    ! Character: O
    PROC char_upperO()
        VAR robtarget pTarget;
        pTarget:=refTarget;
        pTarget.trans:=[12,32.0,0];
        MoveL pTarget,vSpeed,fine,tTool\WObj:=wWobj;
        Set do_pen;
        pTarget.trans:=[9,31.0,0];
        MoveL pTarget,vSpeed,z0,tTool\WObj:=wWobj;
        pTarget.trans:=[7,29.0,0];
        MoveL pTarget,vSpeed,z0,tTool\WObj:=wWobj;
        pTarget.trans:=[5,26.0,0];
        MoveL pTarget,vSpeed,z0,tTool\WObj:=wWobj;
        pTarget.trans:=[4,24.0,0];
        MoveL pTarget,vSpeed,z0,tTool\WObj:=wWobj;
        pTarget.trans:=[3,20.0,0];
        MoveL pTarget,vSpeed,z0,tTool\WObj:=wWobj;
        pTarget.trans:=[3,16.0,0];
        MoveL pTarget,vSpeed,z0,tTool\WObj:=wWobj;
        pTarget.trans:=[4,13.0,0];
        MoveL pTarget,vSpeed,z0,tTool\WObj:=wWobj;
        pTarget.trans:=[5,12.0,0];
        MoveL pTarget,vSpeed,z0,tTool\WObj:=wWobj;
        pTarget.trans:=[7,11.0,0];
        MoveL pTarget,vSpeed,z0,tTool\WObj:=wWobj;
        pTarget.trans:=[9,11.0,0];
        MoveL pTarget,vSpeed,z0,tTool\WObj:=wWobj;
        pTarget.trans:=[12,12.0,0];
        MoveL pTarget,vSpeed,z0,tTool\WObj:=wWobj;
        pTarget.trans:=[14,14.0,0];
        MoveL pTarget,vSpeed,z0,tTool\WObj:=wWobj;
        pTarget.trans:=[16,17.0,0];
        MoveL pTarget,vSpeed,z0,tTool\WObj:=wWobj;
        pTarget.trans:=[17,19.0,0];
        MoveL pTarget,vSpeed,z0,tTool\WObj:=wWobj;
        pTarget.trans:=[18,23.0,0];
        MoveL pTarget,vSpeed,z0,tTool\WObj:=wWobj;
        pTarget.trans:=[18,27.0,0];
        MoveL pTarget,vSpeed,z0,tTool\WObj:=wWobj;
        pTarget.trans:=[17,30.0,0];
        MoveL pTarget,vSpeed,z0,tTool\WObj:=wWobj;
        pTarget.trans:=[16,31.0,0];
        MoveL pTarget,vSpeed,z0,tTool\WObj:=wWobj;
        pTarget.trans:=[14,32.0,0];
        MoveL pTarget,vSpeed,z0,tTool\WObj:=wWobj;
        pTarget.trans:=[12,32.0,0];
        MoveL pTarget,vSpeed,z0,tTool\WObj:=wWobj;
        pTarget.trans:=[10,30.0,0];
        MoveL pTarget,vSpeed,z0,tTool\WObj:=wWobj;
        pTarget.trans:=[10,27.0,0];
        MoveL pTarget,vSpeed,z0,tTool\WObj:=wWobj;
        pTarget.trans:=[11,24.0,0];
        MoveL pTarget,vSpeed,z0,tTool\WObj:=wWobj;
        pTarget.trans:=[13,21.0,0];
        MoveL pTarget,vSpeed,z0,tTool\WObj:=wWobj;
        pTarget.trans:=[15,19.0,0];
        MoveL pTarget,vSpeed,z0,tTool\WObj:=wWobj;
        pTarget.trans:=[18,17.0,0];
        MoveL pTarget,vSpeed,z0,tTool\WObj:=wWobj;
        pTarget.trans:=[20,16.0,0];
        MoveL pTarget,vSpeed,fine,tTool\WObj:=wWobj;
        Reset do_pen;
        MoveL RelTool(pTarget,0,0,-2),vSpeed,z0,tTool\WObj:=wWobj;
        wWobj.oframe.trans.x:=wWobj.oframe.trans.x+17;
    ENDPROC

    ! Character: P
    PROC char_upperP()
        VAR robtarget pTarget;
        pTarget:=refTarget;
        pTarget.trans:=[13,30.0,0];
        MoveL pTarget,vSpeed,fine,tTool\WObj:=wWobj;
        Set do_pen;
        pTarget.trans:=[14,29.0,0];
        MoveL pTarget,vSpeed,z0,tTool\WObj:=wWobj;
        pTarget.trans:=[14,26.0,0];
        MoveL pTarget,vSpeed,z0,tTool\WObj:=wWobj;
        pTarget.trans:=[13,22.0,0];
        MoveL pTarget,vSpeed,z0,tTool\WObj:=wWobj;
        pTarget.trans:=[12,19.0,0];
        MoveL pTarget,vSpeed,z0,tTool\WObj:=wWobj;
        pTarget.trans:=[11,17.0,0];
        MoveL pTarget,vSpeed,z0,tTool\WObj:=wWobj;
        pTarget.trans:=[9,14.0,0];
        MoveL pTarget,vSpeed,z0,tTool\WObj:=wWobj;
        pTarget.trans:=[7,12.0,0];
        MoveL pTarget,vSpeed,z0,tTool\WObj:=wWobj;
        pTarget.trans:=[5,11.0,0];
        MoveL pTarget,vSpeed,z0,tTool\WObj:=wWobj;
        pTarget.trans:=[4,11.0,0];
        MoveL pTarget,vSpeed,z0,tTool\WObj:=wWobj;
        pTarget.trans:=[3,12.0,0];
        MoveL pTarget,vSpeed,z0,tTool\WObj:=wWobj;
        pTarget.trans:=[3,15.0,0];
        MoveL pTarget,vSpeed,z0,tTool\WObj:=wWobj;
        pTarget.trans:=[4,20.0,0];
        MoveL pTarget,vSpeed,z0,tTool\WObj:=wWobj;
        pTarget.trans:=[5,23.0,0];
        MoveL pTarget,vSpeed,z0,tTool\WObj:=wWobj;
        pTarget.trans:=[6,25.0,0];
        MoveL pTarget,vSpeed,z0,tTool\WObj:=wWobj;
        pTarget.trans:=[8,28.0,0];
        MoveL pTarget,vSpeed,z0,tTool\WObj:=wWobj;
        pTarget.trans:=[10,30.0,0];
        MoveL pTarget,vSpeed,z0,tTool\WObj:=wWobj;
        pTarget.trans:=[12,31.0,0];
        MoveL pTarget,vSpeed,z0,tTool\WObj:=wWobj;
        pTarget.trans:=[15,32.0,0];
        MoveL pTarget,vSpeed,z0,tTool\WObj:=wWobj;
        pTarget.trans:=[20,32.0,0];
        MoveL pTarget,vSpeed,z0,tTool\WObj:=wWobj;
        pTarget.trans:=[22,31.0,0];
        MoveL pTarget,vSpeed,z0,tTool\WObj:=wWobj;
        pTarget.trans:=[23,30.0,0];
        MoveL pTarget,vSpeed,z0,tTool\WObj:=wWobj;
        pTarget.trans:=[24,28.0,0];
        MoveL pTarget,vSpeed,z0,tTool\WObj:=wWobj;
        pTarget.trans:=[24,25.0,0];
        MoveL pTarget,vSpeed,z0,tTool\WObj:=wWobj;
        pTarget.trans:=[23,23.0,0];
        MoveL pTarget,vSpeed,z0,tTool\WObj:=wWobj;
        pTarget.trans:=[22,22.0,0];
        MoveL pTarget,vSpeed,z0,tTool\WObj:=wWobj;
        pTarget.trans:=[20,21.0,0];
        MoveL pTarget,vSpeed,z0,tTool\WObj:=wWobj;
        pTarget.trans:=[17,21.0,0];
        MoveL pTarget,vSpeed,z0,tTool\WObj:=wWobj;
        pTarget.trans:=[15,22.0,0];
        MoveL pTarget,vSpeed,z0,tTool\WObj:=wWobj;
        pTarget.trans:=[14,23.0,0];
        MoveL pTarget,vSpeed,fine,tTool\WObj:=wWobj;
        Reset do_pen;
        MoveL RelTool(pTarget,0,0,-2),vSpeed,z0,tTool\WObj:=wWobj;
        wWobj.oframe.trans.x:=wWobj.oframe.trans.x+21;
    ENDPROC

    ! Character: Q
    PROC char_upperQ()
        VAR robtarget pTarget;
        pTarget:=refTarget;
        pTarget.trans:=[13,26.0,0];
        MoveL pTarget,vSpeed,fine,tTool\WObj:=wWobj;
        Set do_pen;
        pTarget.trans:=[12,24.0,0];
        MoveL pTarget,vSpeed,z0,tTool\WObj:=wWobj;
        pTarget.trans:=[11,23.0,0];
        MoveL pTarget,vSpeed,z0,tTool\WObj:=wWobj;
        pTarget.trans:=[9,22.0,0];
        MoveL pTarget,vSpeed,z0,tTool\WObj:=wWobj;
        pTarget.trans:=[7,22.0,0];
        MoveL pTarget,vSpeed,z0,tTool\WObj:=wWobj;
        pTarget.trans:=[6,24.0,0];
        MoveL pTarget,vSpeed,z0,tTool\WObj:=wWobj;
        pTarget.trans:=[6,26.0,0];
        MoveL pTarget,vSpeed,z0,tTool\WObj:=wWobj;
        pTarget.trans:=[7,29.0,0];
        MoveL pTarget,vSpeed,z0,tTool\WObj:=wWobj;
        pTarget.trans:=[9,31.0,0];
        MoveL pTarget,vSpeed,z0,tTool\WObj:=wWobj;
        pTarget.trans:=[12,32.0,0];
        MoveL pTarget,vSpeed,z0,tTool\WObj:=wWobj;
        pTarget.trans:=[15,32.0,0];
        MoveL pTarget,vSpeed,z0,tTool\WObj:=wWobj;
        pTarget.trans:=[17,31.0,0];
        MoveL pTarget,vSpeed,z0,tTool\WObj:=wWobj;
        pTarget.trans:=[18,29.0,0];
        MoveL pTarget,vSpeed,z0,tTool\WObj:=wWobj;
        pTarget.trans:=[18,25.0,0];
        MoveL pTarget,vSpeed,z0,tTool\WObj:=wWobj;
        pTarget.trans:=[17,22.0,0];
        MoveL pTarget,vSpeed,z0,tTool\WObj:=wWobj;
        pTarget.trans:=[15,19.0,0];
        MoveL pTarget,vSpeed,z0,tTool\WObj:=wWobj;
        pTarget.trans:=[11,15.0,0];
        MoveL pTarget,vSpeed,z0,tTool\WObj:=wWobj;
        pTarget.trans:=[8,13.0,0];
        MoveL pTarget,vSpeed,z0,tTool\WObj:=wWobj;
        pTarget.trans:=[6,12.0,0];
        MoveL pTarget,vSpeed,z0,tTool\WObj:=wWobj;
        pTarget.trans:=[3,11.0,0];
        MoveL pTarget,vSpeed,z0,tTool\WObj:=wWobj;
        pTarget.trans:=[1,11.0,0];
        MoveL pTarget,vSpeed,z0,tTool\WObj:=wWobj;
        pTarget.trans:=[0,12.0,0];
        MoveL pTarget,vSpeed,z0,tTool\WObj:=wWobj;
        pTarget.trans:=[0,14.0,0];
        MoveL pTarget,vSpeed,z0,tTool\WObj:=wWobj;
        pTarget.trans:=[1,15.0,0];
        MoveL pTarget,vSpeed,z0,tTool\WObj:=wWobj;
        pTarget.trans:=[3,15.0,0];
        MoveL pTarget,vSpeed,z0,tTool\WObj:=wWobj;
        pTarget.trans:=[5,14.0,0];
        MoveL pTarget,vSpeed,z0,tTool\WObj:=wWobj;
        pTarget.trans:=[8,12.0,0];
        MoveL pTarget,vSpeed,z0,tTool\WObj:=wWobj;
        pTarget.trans:=[11,11.0,0];
        MoveL pTarget,vSpeed,z0,tTool\WObj:=wWobj;
        pTarget.trans:=[14,11.0,0];
        MoveL pTarget,vSpeed,z0,tTool\WObj:=wWobj;
        pTarget.trans:=[17,12.0,0];
        MoveL pTarget,vSpeed,z0,tTool\WObj:=wWobj;
        pTarget.trans:=[19,14.0,0];
        MoveL pTarget,vSpeed,fine,tTool\WObj:=wWobj;
        Reset do_pen;
        MoveL RelTool(pTarget,0,0,-2),vSpeed,z0,tTool\WObj:=wWobj;
        wWobj.oframe.trans.x:=wWobj.oframe.trans.x+19;
    ENDPROC

    ! Character: R
    PROC char_upperR()
        VAR robtarget pTarget;
        pTarget:=refTarget;
        pTarget.trans:=[13,30.0,0];
        MoveL pTarget,vSpeed,fine,tTool\WObj:=wWobj;
        Set do_pen;
        pTarget.trans:=[14,29.0,0];
        MoveL pTarget,vSpeed,z0,tTool\WObj:=wWobj;
        pTarget.trans:=[14,26.0,0];
        MoveL pTarget,vSpeed,z0,tTool\WObj:=wWobj;
        pTarget.trans:=[13,22.0,0];
        MoveL pTarget,vSpeed,z0,tTool\WObj:=wWobj;
        pTarget.trans:=[12,19.0,0];
        MoveL pTarget,vSpeed,z0,tTool\WObj:=wWobj;
        pTarget.trans:=[11,17.0,0];
        MoveL pTarget,vSpeed,z0,tTool\WObj:=wWobj;
        pTarget.trans:=[9,14.0,0];
        MoveL pTarget,vSpeed,z0,tTool\WObj:=wWobj;
        pTarget.trans:=[7,12.0,0];
        MoveL pTarget,vSpeed,z0,tTool\WObj:=wWobj;
        pTarget.trans:=[5,11.0,0];
        MoveL pTarget,vSpeed,z0,tTool\WObj:=wWobj;
        pTarget.trans:=[4,11.0,0];
        MoveL pTarget,vSpeed,z0,tTool\WObj:=wWobj;
        pTarget.trans:=[3,12.0,0];
        MoveL pTarget,vSpeed,z0,tTool\WObj:=wWobj;
        pTarget.trans:=[3,15.0,0];
        MoveL pTarget,vSpeed,z0,tTool\WObj:=wWobj;
        pTarget.trans:=[4,20.0,0];
        MoveL pTarget,vSpeed,z0,tTool\WObj:=wWobj;
        pTarget.trans:=[5,23.0,0];
        MoveL pTarget,vSpeed,z0,tTool\WObj:=wWobj;
        pTarget.trans:=[6,25.0,0];
        MoveL pTarget,vSpeed,z0,tTool\WObj:=wWobj;
        pTarget.trans:=[8,28.0,0];
        MoveL pTarget,vSpeed,z0,tTool\WObj:=wWobj;
        pTarget.trans:=[10,30.0,0];
        MoveL pTarget,vSpeed,z0,tTool\WObj:=wWobj;
        pTarget.trans:=[12,31.0,0];
        MoveL pTarget,vSpeed,z0,tTool\WObj:=wWobj;
        pTarget.trans:=[15,32.0,0];
        MoveL pTarget,vSpeed,z0,tTool\WObj:=wWobj;
        pTarget.trans:=[19,32.0,0];
        MoveL pTarget,vSpeed,z0,tTool\WObj:=wWobj;
        pTarget.trans:=[21,31.0,0];
        MoveL pTarget,vSpeed,z0,tTool\WObj:=wWobj;
        pTarget.trans:=[22,30.0,0];
        MoveL pTarget,vSpeed,z0,tTool\WObj:=wWobj;
        pTarget.trans:=[23,28.0,0];
        MoveL pTarget,vSpeed,z0,tTool\WObj:=wWobj;
        pTarget.trans:=[23,25.0,0];
        MoveL pTarget,vSpeed,z0,tTool\WObj:=wWobj;
        pTarget.trans:=[22,23.0,0];
        MoveL pTarget,vSpeed,z0,tTool\WObj:=wWobj;
        pTarget.trans:=[21,22.0,0];
        MoveL pTarget,vSpeed,z0,tTool\WObj:=wWobj;
        pTarget.trans:=[19,21.0,0];
        MoveL pTarget,vSpeed,z0,tTool\WObj:=wWobj;
        pTarget.trans:=[16,21.0,0];
        MoveL pTarget,vSpeed,z0,tTool\WObj:=wWobj;
        pTarget.trans:=[13,22.0,0];
        MoveL pTarget,vSpeed,z0,tTool\WObj:=wWobj;
        pTarget.trans:=[14,21.0,0];
        MoveL pTarget,vSpeed,z0,tTool\WObj:=wWobj;
        pTarget.trans:=[15,19.0,0];
        MoveL pTarget,vSpeed,z0,tTool\WObj:=wWobj;
        pTarget.trans:=[15,14.0,0];
        MoveL pTarget,vSpeed,z0,tTool\WObj:=wWobj;
        pTarget.trans:=[16,12.0,0];
        MoveL pTarget,vSpeed,z0,tTool\WObj:=wWobj;
        pTarget.trans:=[18,11.0,0];
        MoveL pTarget,vSpeed,z0,tTool\WObj:=wWobj;
        pTarget.trans:=[20,12.0,0];
        MoveL pTarget,vSpeed,z0,tTool\WObj:=wWobj;
        pTarget.trans:=[21,13.0,0];
        MoveL pTarget,vSpeed,z0,tTool\WObj:=wWobj;
        pTarget.trans:=[23,16.0,0];
        MoveL pTarget,vSpeed,fine,tTool\WObj:=wWobj;
        Reset do_pen;
        MoveL RelTool(pTarget,0,0,-2),vSpeed,z0,tTool\WObj:=wWobj;
        wWobj.oframe.trans.x:=wWobj.oframe.trans.x+20;
    ENDPROC

    ! Character: S
    PROC char_upperS()
        VAR robtarget pTarget;
        pTarget:=refTarget;
        pTarget.trans:=[0,11.0,0];
        MoveL pTarget,vSpeed,fine,tTool\WObj:=wWobj;
        Set do_pen;
        pTarget.trans:=[2,12.0,0];
        MoveL pTarget,vSpeed,z0,tTool\WObj:=wWobj;
        pTarget.trans:=[4,14.0,0];
        MoveL pTarget,vSpeed,z0,tTool\WObj:=wWobj;
        pTarget.trans:=[7,18.0,0];
        MoveL pTarget,vSpeed,z0,tTool\WObj:=wWobj;
        pTarget.trans:=[9,21.0,0];
        MoveL pTarget,vSpeed,z0,tTool\WObj:=wWobj;
        pTarget.trans:=[11,25.0,0];
        MoveL pTarget,vSpeed,z0,tTool\WObj:=wWobj;
        pTarget.trans:=[12,28.0,0];
        MoveL pTarget,vSpeed,z0,tTool\WObj:=wWobj;
        pTarget.trans:=[12,31.0,0];
        MoveL pTarget,vSpeed,z0,tTool\WObj:=wWobj;
        pTarget.trans:=[11,32.0,0];
        MoveL pTarget,vSpeed,z0,tTool\WObj:=wWobj;
        pTarget.trans:=[10,32.0,0];
        MoveL pTarget,vSpeed,z0,tTool\WObj:=wWobj;
        pTarget.trans:=[9,31.0,0];
        MoveL pTarget,vSpeed,z0,tTool\WObj:=wWobj;
        pTarget.trans:=[8,29.0,0];
        MoveL pTarget,vSpeed,z0,tTool\WObj:=wWobj;
        pTarget.trans:=[8,27.0,0];
        MoveL pTarget,vSpeed,z0,tTool\WObj:=wWobj;
        pTarget.trans:=[9,25.0,0];
        MoveL pTarget,vSpeed,z0,tTool\WObj:=wWobj;
        pTarget.trans:=[11,23.0,0];
        MoveL pTarget,vSpeed,z0,tTool\WObj:=wWobj;
        pTarget.trans:=[14,21.0,0];
        MoveL pTarget,vSpeed,z0,tTool\WObj:=wWobj;
        pTarget.trans:=[16,19.0,0];
        MoveL pTarget,vSpeed,z0,tTool\WObj:=wWobj;
        pTarget.trans:=[17,17.0,0];
        MoveL pTarget,vSpeed,z0,tTool\WObj:=wWobj;
        pTarget.trans:=[17,15.0,0];
        MoveL pTarget,vSpeed,z0,tTool\WObj:=wWobj;
        pTarget.trans:=[16,13.0,0];
        MoveL pTarget,vSpeed,z0,tTool\WObj:=wWobj;
        pTarget.trans:=[15,12.0,0];
        MoveL pTarget,vSpeed,z0,tTool\WObj:=wWobj;
        pTarget.trans:=[12,11.0,0];
        MoveL pTarget,vSpeed,z0,tTool\WObj:=wWobj;
        pTarget.trans:=[8,11.0,0];
        MoveL pTarget,vSpeed,z0,tTool\WObj:=wWobj;
        pTarget.trans:=[5,12.0,0];
        MoveL pTarget,vSpeed,z0,tTool\WObj:=wWobj;
        pTarget.trans:=[3,14.0,0];
        MoveL pTarget,vSpeed,z0,tTool\WObj:=wWobj;
        pTarget.trans:=[2,16.0,0];
        MoveL pTarget,vSpeed,z0,tTool\WObj:=wWobj;
        pTarget.trans:=[2,18.0,0];
        MoveL pTarget,vSpeed,fine,tTool\WObj:=wWobj;
        Reset do_pen;
        MoveL RelTool(pTarget,0,0,-2),vSpeed,z0,tTool\WObj:=wWobj;
        wWobj.oframe.trans.x:=wWobj.oframe.trans.x+17;
    ENDPROC

    ! Character: T
    PROC char_upperT()
        VAR robtarget pTarget;
        pTarget:=refTarget;
        pTarget.trans:=[10,26.0,0];
        MoveL pTarget,vSpeed,fine,tTool\WObj:=wWobj;
        Set do_pen;
        pTarget.trans:=[8,26.0,0];
        MoveL pTarget,vSpeed,z0,tTool\WObj:=wWobj;
        pTarget.trans:=[6,27.0,0];
        MoveL pTarget,vSpeed,z0,tTool\WObj:=wWobj;
        pTarget.trans:=[5,29.0,0];
        MoveL pTarget,vSpeed,z0,tTool\WObj:=wWobj;
        pTarget.trans:=[6,31.0,0];
        MoveL pTarget,vSpeed,z0,tTool\WObj:=wWobj;
        pTarget.trans:=[9,32.0,0];
        MoveL pTarget,vSpeed,z0,tTool\WObj:=wWobj;
        pTarget.trans:=[12,32.0,0];
        MoveL pTarget,vSpeed,z0,tTool\WObj:=wWobj;
        pTarget.trans:=[16,31.0,0];
        MoveL pTarget,vSpeed,z0,tTool\WObj:=wWobj;
        pTarget.trans:=[19,31.0,0];
        MoveL pTarget,vSpeed,z0,tTool\WObj:=wWobj;
        pTarget.trans:=[21,32.0,0];
        MoveL pTarget,vSpeed,fine,tTool\WObj:=wWobj;
        Reset do_pen;
        MoveL RelTool(pTarget,0,0,-2),vSpeed,z0,tTool\WObj:=wWobj;
        pTarget.trans:=[16,31.0,0];
        MoveL pTarget,vSpeed,fine,tTool\WObj:=wWobj;
        Set do_pen;
        pTarget.trans:=[14,24.0,0];
        MoveL pTarget,vSpeed,z0,tTool\WObj:=wWobj;
        pTarget.trans:=[12,18.0,0];
        MoveL pTarget,vSpeed,z0,tTool\WObj:=wWobj;
        pTarget.trans:=[10,14.0,0];
        MoveL pTarget,vSpeed,z0,tTool\WObj:=wWobj;
        pTarget.trans:=[8,12.0,0];
        MoveL pTarget,vSpeed,z0,tTool\WObj:=wWobj;
        pTarget.trans:=[6,11.0,0];
        MoveL pTarget,vSpeed,z0,tTool\WObj:=wWobj;
        pTarget.trans:=[4,11.0,0];
        MoveL pTarget,vSpeed,z0,tTool\WObj:=wWobj;
        pTarget.trans:=[2,12.0,0];
        MoveL pTarget,vSpeed,z0,tTool\WObj:=wWobj;
        pTarget.trans:=[1,14.0,0];
        MoveL pTarget,vSpeed,z0,tTool\WObj:=wWobj;
        pTarget.trans:=[1,16.0,0];
        MoveL pTarget,vSpeed,z0,tTool\WObj:=wWobj;
        pTarget.trans:=[2,17.0,0];
        MoveL pTarget,vSpeed,z0,tTool\WObj:=wWobj;
        pTarget.trans:=[4,17.0,0];
        MoveL pTarget,vSpeed,z0,tTool\WObj:=wWobj;
        pTarget.trans:=[6,16.0,0];
        MoveL pTarget,vSpeed,fine,tTool\WObj:=wWobj;
        Reset do_pen;
        MoveL RelTool(pTarget,0,0,-2),vSpeed,z0,tTool\WObj:=wWobj;
        wWobj.oframe.trans.x:=wWobj.oframe.trans.x+20;
    ENDPROC

    ! Character: U
    PROC char_upperU()
        VAR robtarget pTarget;
        pTarget:=refTarget;
        pTarget.trans:=[5,25.0,0];
        MoveL pTarget,vSpeed,fine,tTool\WObj:=wWobj;
        Set do_pen;
        pTarget.trans:=[3,26.0,0];
        MoveL pTarget,vSpeed,z0,tTool\WObj:=wWobj;
        pTarget.trans:=[2,28.0,0];
        MoveL pTarget,vSpeed,z0,tTool\WObj:=wWobj;
        pTarget.trans:=[2,29.0,0];
        MoveL pTarget,vSpeed,z0,tTool\WObj:=wWobj;
        pTarget.trans:=[3,31.0,0];
        MoveL pTarget,vSpeed,z0,tTool\WObj:=wWobj;
        pTarget.trans:=[5,32.0,0];
        MoveL pTarget,vSpeed,z0,tTool\WObj:=wWobj;
        pTarget.trans:=[6,32.0,0];
        MoveL pTarget,vSpeed,z0,tTool\WObj:=wWobj;
        pTarget.trans:=[8,31.0,0];
        MoveL pTarget,vSpeed,z0,tTool\WObj:=wWobj;
        pTarget.trans:=[9,29.0,0];
        MoveL pTarget,vSpeed,z0,tTool\WObj:=wWobj;
        pTarget.trans:=[9,27.0,0];
        MoveL pTarget,vSpeed,z0,tTool\WObj:=wWobj;
        pTarget.trans:=[8,23.0,0];
        MoveL pTarget,vSpeed,z0,tTool\WObj:=wWobj;
        pTarget.trans:=[7,20.0,0];
        MoveL pTarget,vSpeed,z0,tTool\WObj:=wWobj;
        pTarget.trans:=[6,16.0,0];
        MoveL pTarget,vSpeed,z0,tTool\WObj:=wWobj;
        pTarget.trans:=[6,14.0,0];
        MoveL pTarget,vSpeed,z0,tTool\WObj:=wWobj;
        pTarget.trans:=[7,12.0,0];
        MoveL pTarget,vSpeed,z0,tTool\WObj:=wWobj;
        pTarget.trans:=[9,11.0,0];
        MoveL pTarget,vSpeed,z0,tTool\WObj:=wWobj;
        pTarget.trans:=[11,11.0,0];
        MoveL pTarget,vSpeed,z0,tTool\WObj:=wWobj;
        pTarget.trans:=[13,12.0,0];
        MoveL pTarget,vSpeed,z0,tTool\WObj:=wWobj;
        pTarget.trans:=[14,13.0,0];
        MoveL pTarget,vSpeed,z0,tTool\WObj:=wWobj;
        pTarget.trans:=[16,17.0,0];
        MoveL pTarget,vSpeed,z0,tTool\WObj:=wWobj;
        pTarget.trans:=[19,25.0,0];
        MoveL pTarget,vSpeed,z0,tTool\WObj:=wWobj;
        pTarget.trans:=[21,32.0,0];
        MoveL pTarget,vSpeed,fine,tTool\WObj:=wWobj;
        Reset do_pen;
        MoveL RelTool(pTarget,0,0,-2),vSpeed,z0,tTool\WObj:=wWobj;
        pTarget.trans:=[19,25.0,0];
        MoveL pTarget,vSpeed,fine,tTool\WObj:=wWobj;
        Set do_pen;
        pTarget.trans:=[18,21.0,0];
        MoveL pTarget,vSpeed,z0,tTool\WObj:=wWobj;
        pTarget.trans:=[17,15.0,0];
        MoveL pTarget,vSpeed,z0,tTool\WObj:=wWobj;
        pTarget.trans:=[17,12.0,0];
        MoveL pTarget,vSpeed,z0,tTool\WObj:=wWobj;
        pTarget.trans:=[18,11.0,0];
        MoveL pTarget,vSpeed,z0,tTool\WObj:=wWobj;
        pTarget.trans:=[19,11.0,0];
        MoveL pTarget,vSpeed,z0,tTool\WObj:=wWobj;
        pTarget.trans:=[21,12.0,0];
        MoveL pTarget,vSpeed,z0,tTool\WObj:=wWobj;
        pTarget.trans:=[22,13.0,0];
        MoveL pTarget,vSpeed,z0,tTool\WObj:=wWobj;
        pTarget.trans:=[24,16.0,0];
        MoveL pTarget,vSpeed,fine,tTool\WObj:=wWobj;
        Reset do_pen;
        MoveL RelTool(pTarget,0,0,-2),vSpeed,z0,tTool\WObj:=wWobj;
        wWobj.oframe.trans.x:=wWobj.oframe.trans.x+22;
    ENDPROC

    ! Character: V
    PROC char_upperV()
        VAR robtarget pTarget;
        pTarget:=refTarget;
        pTarget.trans:=[5,25.0,0];
        MoveL pTarget,vSpeed,fine,tTool\WObj:=wWobj;
        Set do_pen;
        pTarget.trans:=[3,26.0,0];
        MoveL pTarget,vSpeed,z0,tTool\WObj:=wWobj;
        pTarget.trans:=[2,28.0,0];
        MoveL pTarget,vSpeed,z0,tTool\WObj:=wWobj;
        pTarget.trans:=[2,29.0,0];
        MoveL pTarget,vSpeed,z0,tTool\WObj:=wWobj;
        pTarget.trans:=[3,31.0,0];
        MoveL pTarget,vSpeed,z0,tTool\WObj:=wWobj;
        pTarget.trans:=[5,32.0,0];
        MoveL pTarget,vSpeed,z0,tTool\WObj:=wWobj;
        pTarget.trans:=[6,32.0,0];
        MoveL pTarget,vSpeed,z0,tTool\WObj:=wWobj;
        pTarget.trans:=[8,31.0,0];
        MoveL pTarget,vSpeed,z0,tTool\WObj:=wWobj;
        pTarget.trans:=[9,29.0,0];
        MoveL pTarget,vSpeed,z0,tTool\WObj:=wWobj;
        pTarget.trans:=[9,27.0,0];
        MoveL pTarget,vSpeed,z0,tTool\WObj:=wWobj;
        pTarget.trans:=[8,23.0,0];
        MoveL pTarget,vSpeed,z0,tTool\WObj:=wWobj;
        pTarget.trans:=[7,20.0,0];
        MoveL pTarget,vSpeed,z0,tTool\WObj:=wWobj;
        pTarget.trans:=[6,16.0,0];
        MoveL pTarget,vSpeed,z0,tTool\WObj:=wWobj;
        pTarget.trans:=[6,13.0,0];
        MoveL pTarget,vSpeed,z0,tTool\WObj:=wWobj;
        pTarget.trans:=[7,11.0,0];
        MoveL pTarget,vSpeed,z0,tTool\WObj:=wWobj;
        pTarget.trans:=[9,11.0,0];
        MoveL pTarget,vSpeed,z0,tTool\WObj:=wWobj;
        pTarget.trans:=[11,12.0,0];
        MoveL pTarget,vSpeed,z0,tTool\WObj:=wWobj;
        pTarget.trans:=[14,15.0,0];
        MoveL pTarget,vSpeed,z0,tTool\WObj:=wWobj;
        pTarget.trans:=[16,18.0,0];
        MoveL pTarget,vSpeed,z0,tTool\WObj:=wWobj;
        pTarget.trans:=[18,22.0,0];
        MoveL pTarget,vSpeed,z0,tTool\WObj:=wWobj;
        pTarget.trans:=[19,25.0,0];
        MoveL pTarget,vSpeed,z0,tTool\WObj:=wWobj;
        pTarget.trans:=[20,29.0,0];
        MoveL pTarget,vSpeed,z0,tTool\WObj:=wWobj;
        pTarget.trans:=[20,31.0,0];
        MoveL pTarget,vSpeed,z0,tTool\WObj:=wWobj;
        pTarget.trans:=[19,32.0,0];
        MoveL pTarget,vSpeed,z0,tTool\WObj:=wWobj;
        pTarget.trans:=[18,32.0,0];
        MoveL pTarget,vSpeed,z0,tTool\WObj:=wWobj;
        pTarget.trans:=[17,31.0,0];
        MoveL pTarget,vSpeed,z0,tTool\WObj:=wWobj;
        pTarget.trans:=[16,29.0,0];
        MoveL pTarget,vSpeed,z0,tTool\WObj:=wWobj;
        pTarget.trans:=[16,27.0,0];
        MoveL pTarget,vSpeed,z0,tTool\WObj:=wWobj;
        pTarget.trans:=[17,24.0,0];
        MoveL pTarget,vSpeed,z0,tTool\WObj:=wWobj;
        pTarget.trans:=[19,22.0,0];
        MoveL pTarget,vSpeed,z0,tTool\WObj:=wWobj;
        pTarget.trans:=[21,21.0,0];
        MoveL pTarget,vSpeed,fine,tTool\WObj:=wWobj;
        Reset do_pen;
        MoveL RelTool(pTarget,0,0,-2),vSpeed,z0,tTool\WObj:=wWobj;
        wWobj.oframe.trans.x:=wWobj.oframe.trans.x+19;
    ENDPROC

    ! Character: W
    PROC char_upperW()
        VAR robtarget pTarget;
        pTarget:=refTarget;
        pTarget.trans:=[5,25.0,0];
        MoveL pTarget,vSpeed,fine,tTool\WObj:=wWobj;
        Set do_pen;
        pTarget.trans:=[3,26.0,0];
        MoveL pTarget,vSpeed,z0,tTool\WObj:=wWobj;
        pTarget.trans:=[2,28.0,0];
        MoveL pTarget,vSpeed,z0,tTool\WObj:=wWobj;
        pTarget.trans:=[2,29.0,0];
        MoveL pTarget,vSpeed,z0,tTool\WObj:=wWobj;
        pTarget.trans:=[3,31.0,0];
        MoveL pTarget,vSpeed,z0,tTool\WObj:=wWobj;
        pTarget.trans:=[5,32.0,0];
        MoveL pTarget,vSpeed,z0,tTool\WObj:=wWobj;
        pTarget.trans:=[6,32.0,0];
        MoveL pTarget,vSpeed,z0,tTool\WObj:=wWobj;
        pTarget.trans:=[8,31.0,0];
        MoveL pTarget,vSpeed,z0,tTool\WObj:=wWobj;
        pTarget.trans:=[9,29.0,0];
        MoveL pTarget,vSpeed,z0,tTool\WObj:=wWobj;
        pTarget.trans:=[9,26.0,0];
        MoveL pTarget,vSpeed,z0,tTool\WObj:=wWobj;
        pTarget.trans:=[8,11.0,0];
        MoveL pTarget,vSpeed,fine,tTool\WObj:=wWobj;
        Reset do_pen;
        MoveL RelTool(pTarget,0,0,-2),vSpeed,z0,tTool\WObj:=wWobj;
        pTarget.trans:=[18,32.0,0];
        MoveL pTarget,vSpeed,fine,tTool\WObj:=wWobj;
        Set do_pen;
        pTarget.trans:=[8,11.0,0];
        MoveL pTarget,vSpeed,fine,tTool\WObj:=wWobj;
        Reset do_pen;
        MoveL RelTool(pTarget,0,0,-2),vSpeed,z0,tTool\WObj:=wWobj;
        pTarget.trans:=[18,32.0,0];
        MoveL pTarget,vSpeed,fine,tTool\WObj:=wWobj;
        Set do_pen;
        pTarget.trans:=[16,11.0,0];
        MoveL pTarget,vSpeed,fine,tTool\WObj:=wWobj;
        Reset do_pen;
        MoveL RelTool(pTarget,0,0,-2),vSpeed,z0,tTool\WObj:=wWobj;
        pTarget.trans:=[30,32.0,0];
        MoveL pTarget,vSpeed,fine,tTool\WObj:=wWobj;
        Set do_pen;
        pTarget.trans:=[28,31.0,0];
        MoveL pTarget,vSpeed,z0,tTool\WObj:=wWobj;
        pTarget.trans:=[25,28.0,0];
        MoveL pTarget,vSpeed,z0,tTool\WObj:=wWobj;
        pTarget.trans:=[22,24.0,0];
        MoveL pTarget,vSpeed,z0,tTool\WObj:=wWobj;
        pTarget.trans:=[19,18.0,0];
        MoveL pTarget,vSpeed,z0,tTool\WObj:=wWobj;
        pTarget.trans:=[16,11.0,0];
        MoveL pTarget,vSpeed,fine,tTool\WObj:=wWobj;
        Reset do_pen;
        MoveL RelTool(pTarget,0,0,-2),vSpeed,z0,tTool\WObj:=wWobj;
        wWobj.oframe.trans.x:=wWobj.oframe.trans.x+28;
    ENDPROC

    ! Character: X
    PROC char_upperX()
        VAR robtarget pTarget;
        pTarget:=refTarget;
        pTarget.trans:=[8,26.0,0];
        MoveL pTarget,vSpeed,fine,tTool\WObj:=wWobj;
        Set do_pen;
        pTarget.trans:=[6,26.0,0];
        MoveL pTarget,vSpeed,z0,tTool\WObj:=wWobj;
        pTarget.trans:=[5,27.0,0];
        MoveL pTarget,vSpeed,z0,tTool\WObj:=wWobj;
        pTarget.trans:=[5,29.0,0];
        MoveL pTarget,vSpeed,z0,tTool\WObj:=wWobj;
        pTarget.trans:=[6,31.0,0];
        MoveL pTarget,vSpeed,z0,tTool\WObj:=wWobj;
        pTarget.trans:=[8,32.0,0];
        MoveL pTarget,vSpeed,z0,tTool\WObj:=wWobj;
        pTarget.trans:=[10,32.0,0];
        MoveL pTarget,vSpeed,z0,tTool\WObj:=wWobj;
        pTarget.trans:=[12,31.0,0];
        MoveL pTarget,vSpeed,z0,tTool\WObj:=wWobj;
        pTarget.trans:=[13,29.0,0];
        MoveL pTarget,vSpeed,z0,tTool\WObj:=wWobj;
        pTarget.trans:=[13,26.0,0];
        MoveL pTarget,vSpeed,z0,tTool\WObj:=wWobj;
        pTarget.trans:=[11,17.0,0];
        MoveL pTarget,vSpeed,z0,tTool\WObj:=wWobj;
        pTarget.trans:=[11,14.0,0];
        MoveL pTarget,vSpeed,z0,tTool\WObj:=wWobj;
        pTarget.trans:=[12,12.0,0];
        MoveL pTarget,vSpeed,z0,tTool\WObj:=wWobj;
        pTarget.trans:=[14,11.0,0];
        MoveL pTarget,vSpeed,z0,tTool\WObj:=wWobj;
        pTarget.trans:=[16,11.0,0];
        MoveL pTarget,vSpeed,z0,tTool\WObj:=wWobj;
        pTarget.trans:=[18,12.0,0];
        MoveL pTarget,vSpeed,z0,tTool\WObj:=wWobj;
        pTarget.trans:=[19,14.0,0];
        MoveL pTarget,vSpeed,z0,tTool\WObj:=wWobj;
        pTarget.trans:=[19,16.0,0];
        MoveL pTarget,vSpeed,z0,tTool\WObj:=wWobj;
        pTarget.trans:=[18,17.0,0];
        MoveL pTarget,vSpeed,z0,tTool\WObj:=wWobj;
        pTarget.trans:=[16,17.0,0];
        MoveL pTarget,vSpeed,fine,tTool\WObj:=wWobj;
        Reset do_pen;
        MoveL RelTool(pTarget,0,0,-2),vSpeed,z0,tTool\WObj:=wWobj;
        pTarget.trans:=[23,29.0,0];
        MoveL pTarget,vSpeed,fine,tTool\WObj:=wWobj;
        Set do_pen;
        pTarget.trans:=[23,31.0,0];
        MoveL pTarget,vSpeed,z0,tTool\WObj:=wWobj;
        pTarget.trans:=[22,32.0,0];
        MoveL pTarget,vSpeed,z0,tTool\WObj:=wWobj;
        pTarget.trans:=[20,32.0,0];
        MoveL pTarget,vSpeed,z0,tTool\WObj:=wWobj;
        pTarget.trans:=[18,31.0,0];
        MoveL pTarget,vSpeed,z0,tTool\WObj:=wWobj;
        pTarget.trans:=[16,29.0,0];
        MoveL pTarget,vSpeed,z0,tTool\WObj:=wWobj;
        pTarget.trans:=[14,26.0,0];
        MoveL pTarget,vSpeed,z0,tTool\WObj:=wWobj;
        pTarget.trans:=[10,17.0,0];
        MoveL pTarget,vSpeed,z0,tTool\WObj:=wWobj;
        pTarget.trans:=[8,14.0,0];
        MoveL pTarget,vSpeed,z0,tTool\WObj:=wWobj;
        pTarget.trans:=[6,12.0,0];
        MoveL pTarget,vSpeed,z0,tTool\WObj:=wWobj;
        pTarget.trans:=[4,11.0,0];
        MoveL pTarget,vSpeed,z0,tTool\WObj:=wWobj;
        pTarget.trans:=[2,11.0,0];
        MoveL pTarget,vSpeed,z0,tTool\WObj:=wWobj;
        pTarget.trans:=[1,12.0,0];
        MoveL pTarget,vSpeed,z0,tTool\WObj:=wWobj;
        pTarget.trans:=[1,14.0,0];
        MoveL pTarget,vSpeed,fine,tTool\WObj:=wWobj;
        Reset do_pen;
        MoveL RelTool(pTarget,0,0,-2),vSpeed,z0,tTool\WObj:=wWobj;
        wWobj.oframe.trans.x:=wWobj.oframe.trans.x+22;
    ENDPROC

    ! Character: Y
    PROC char_upperY()
        VAR robtarget pTarget;
        pTarget:=refTarget;
        pTarget.trans:=[5,25.0,0];
        MoveL pTarget,vSpeed,fine,tTool\WObj:=wWobj;
        Set do_pen;
        pTarget.trans:=[3,26.0,0];
        MoveL pTarget,vSpeed,z0,tTool\WObj:=wWobj;
        pTarget.trans:=[2,28.0,0];
        MoveL pTarget,vSpeed,z0,tTool\WObj:=wWobj;
        pTarget.trans:=[2,29.0,0];
        MoveL pTarget,vSpeed,z0,tTool\WObj:=wWobj;
        pTarget.trans:=[3,31.0,0];
        MoveL pTarget,vSpeed,z0,tTool\WObj:=wWobj;
        pTarget.trans:=[5,32.0,0];
        MoveL pTarget,vSpeed,z0,tTool\WObj:=wWobj;
        pTarget.trans:=[6,32.0,0];
        MoveL pTarget,vSpeed,z0,tTool\WObj:=wWobj;
        pTarget.trans:=[8,31.0,0];
        MoveL pTarget,vSpeed,z0,tTool\WObj:=wWobj;
        pTarget.trans:=[9,29.0,0];
        MoveL pTarget,vSpeed,z0,tTool\WObj:=wWobj;
        pTarget.trans:=[9,27.0,0];
        MoveL pTarget,vSpeed,z0,tTool\WObj:=wWobj;
        pTarget.trans:=[8,23.0,0];
        MoveL pTarget,vSpeed,z0,tTool\WObj:=wWobj;
        pTarget.trans:=[7,20.0,0];
        MoveL pTarget,vSpeed,z0,tTool\WObj:=wWobj;
        pTarget.trans:=[6,16.0,0];
        MoveL pTarget,vSpeed,z0,tTool\WObj:=wWobj;
        pTarget.trans:=[6,14.0,0];
        MoveL pTarget,vSpeed,z0,tTool\WObj:=wWobj;
        pTarget.trans:=[7,12.0,0];
        MoveL pTarget,vSpeed,z0,tTool\WObj:=wWobj;
        pTarget.trans:=[8,11.0,0];
        MoveL pTarget,vSpeed,z0,tTool\WObj:=wWobj;
        pTarget.trans:=[10,11.0,0];
        MoveL pTarget,vSpeed,z0,tTool\WObj:=wWobj;
        pTarget.trans:=[12,12.0,0];
        MoveL pTarget,vSpeed,z0,tTool\WObj:=wWobj;
        pTarget.trans:=[14,14.0,0];
        MoveL pTarget,vSpeed,z0,tTool\WObj:=wWobj;
        pTarget.trans:=[16,17.0,0];
        MoveL pTarget,vSpeed,z0,tTool\WObj:=wWobj;
        pTarget.trans:=[17,19.0,0];
        MoveL pTarget,vSpeed,z0,tTool\WObj:=wWobj;
        pTarget.trans:=[19,25.0,0];
        MoveL pTarget,vSpeed,fine,tTool\WObj:=wWobj;
        Reset do_pen;
        MoveL RelTool(pTarget,0,0,-2),vSpeed,z0,tTool\WObj:=wWobj;
        pTarget.trans:=[21,32.0,0];
        MoveL pTarget,vSpeed,fine,tTool\WObj:=wWobj;
        Set do_pen;
        pTarget.trans:=[19,25.0,0];
        MoveL pTarget,vSpeed,z0,tTool\WObj:=wWobj;
        pTarget.trans:=[16,15.0,0];
        MoveL pTarget,vSpeed,z0,tTool\WObj:=wWobj;
        pTarget.trans:=[14,9.0,0];
        MoveL pTarget,vSpeed,z0,tTool\WObj:=wWobj;
        pTarget.trans:=[12,4.0,0];
        MoveL pTarget,vSpeed,z0,tTool\WObj:=wWobj;
        pTarget.trans:=[10,0.0,0];
        MoveL pTarget,vSpeed,z0,tTool\WObj:=wWobj;
        pTarget.trans:=[8,-1.0,0];
        MoveL pTarget,vSpeed,z0,tTool\WObj:=wWobj;
        pTarget.trans:=[7,0.0,0];
        MoveL pTarget,vSpeed,z0,tTool\WObj:=wWobj;
        pTarget.trans:=[7,2.0,0];
        MoveL pTarget,vSpeed,z0,tTool\WObj:=wWobj;
        pTarget.trans:=[8,5.0,0];
        MoveL pTarget,vSpeed,z0,tTool\WObj:=wWobj;
        pTarget.trans:=[10,8.0,0];
        MoveL pTarget,vSpeed,z0,tTool\WObj:=wWobj;
        pTarget.trans:=[13,11.0,0];
        MoveL pTarget,vSpeed,z0,tTool\WObj:=wWobj;
        pTarget.trans:=[16,13.0,0];
        MoveL pTarget,vSpeed,z0,tTool\WObj:=wWobj;
        pTarget.trans:=[21,16.0,0];
        MoveL pTarget,vSpeed,fine,tTool\WObj:=wWobj;
        Reset do_pen;
        MoveL RelTool(pTarget,0,0,-2),vSpeed,z0,tTool\WObj:=wWobj;
        wWobj.oframe.trans.x:=wWobj.oframe.trans.x+19;
    ENDPROC

    ! Character: Z
    PROC char_upperZ()
        VAR robtarget pTarget;
        pTarget:=refTarget;
        pTarget.trans:=[13,26.0,0];
        MoveL pTarget,vSpeed,fine,tTool\WObj:=wWobj;
        Set do_pen;
        pTarget.trans:=[12,24.0,0];
        MoveL pTarget,vSpeed,z0,tTool\WObj:=wWobj;
        pTarget.trans:=[11,23.0,0];
        MoveL pTarget,vSpeed,z0,tTool\WObj:=wWobj;
        pTarget.trans:=[9,22.0,0];
        MoveL pTarget,vSpeed,z0,tTool\WObj:=wWobj;
        pTarget.trans:=[7,22.0,0];
        MoveL pTarget,vSpeed,z0,tTool\WObj:=wWobj;
        pTarget.trans:=[6,24.0,0];
        MoveL pTarget,vSpeed,z0,tTool\WObj:=wWobj;
        pTarget.trans:=[6,26.0,0];
        MoveL pTarget,vSpeed,z0,tTool\WObj:=wWobj;
        pTarget.trans:=[7,29.0,0];
        MoveL pTarget,vSpeed,z0,tTool\WObj:=wWobj;
        pTarget.trans:=[9,31.0,0];
        MoveL pTarget,vSpeed,z0,tTool\WObj:=wWobj;
        pTarget.trans:=[12,32.0,0];
        MoveL pTarget,vSpeed,z0,tTool\WObj:=wWobj;
        pTarget.trans:=[15,32.0,0];
        MoveL pTarget,vSpeed,z0,tTool\WObj:=wWobj;
        pTarget.trans:=[17,31.0,0];
        MoveL pTarget,vSpeed,z0,tTool\WObj:=wWobj;
        pTarget.trans:=[18,29.0,0];
        MoveL pTarget,vSpeed,z0,tTool\WObj:=wWobj;
        pTarget.trans:=[18,25.0,0];
        MoveL pTarget,vSpeed,z0,tTool\WObj:=wWobj;
        pTarget.trans:=[17,22.0,0];
        MoveL pTarget,vSpeed,z0,tTool\WObj:=wWobj;
        pTarget.trans:=[15,18.0,0];
        MoveL pTarget,vSpeed,z0,tTool\WObj:=wWobj;
        pTarget.trans:=[12,15.0,0];
        MoveL pTarget,vSpeed,z0,tTool\WObj:=wWobj;
        pTarget.trans:=[8,12.0,0];
        MoveL pTarget,vSpeed,z0,tTool\WObj:=wWobj;
        pTarget.trans:=[6,11.0,0];
        MoveL pTarget,vSpeed,z0,tTool\WObj:=wWobj;
        pTarget.trans:=[3,11.0,0];
        MoveL pTarget,vSpeed,z0,tTool\WObj:=wWobj;
        pTarget.trans:=[2,12.0,0];
        MoveL pTarget,vSpeed,z0,tTool\WObj:=wWobj;
        pTarget.trans:=[2,14.0,0];
        MoveL pTarget,vSpeed,z0,tTool\WObj:=wWobj;
        pTarget.trans:=[3,15.0,0];
        MoveL pTarget,vSpeed,z0,tTool\WObj:=wWobj;
        pTarget.trans:=[6,15.0,0];
        MoveL pTarget,vSpeed,z0,tTool\WObj:=wWobj;
        pTarget.trans:=[8,14.0,0];
        MoveL pTarget,vSpeed,z0,tTool\WObj:=wWobj;
        pTarget.trans:=[9,13.0,0];
        MoveL pTarget,vSpeed,z0,tTool\WObj:=wWobj;
        pTarget.trans:=[10,11.0,0];
        MoveL pTarget,vSpeed,z0,tTool\WObj:=wWobj;
        pTarget.trans:=[10,8.0,0];
        MoveL pTarget,vSpeed,z0,tTool\WObj:=wWobj;
        pTarget.trans:=[9,5.0,0];
        MoveL pTarget,vSpeed,z0,tTool\WObj:=wWobj;
        pTarget.trans:=[8,3.0,0];
        MoveL pTarget,vSpeed,z0,tTool\WObj:=wWobj;
        pTarget.trans:=[6,0.0,0];
        MoveL pTarget,vSpeed,z0,tTool\WObj:=wWobj;
        pTarget.trans:=[4,-1.0,0];
        MoveL pTarget,vSpeed,z0,tTool\WObj:=wWobj;
        pTarget.trans:=[3,0.0,0];
        MoveL pTarget,vSpeed,z0,tTool\WObj:=wWobj;
        pTarget.trans:=[3,2.0,0];
        MoveL pTarget,vSpeed,z0,tTool\WObj:=wWobj;
        pTarget.trans:=[4,5.0,0];
        MoveL pTarget,vSpeed,z0,tTool\WObj:=wWobj;
        pTarget.trans:=[6,8.0,0];
        MoveL pTarget,vSpeed,z0,tTool\WObj:=wWobj;
        pTarget.trans:=[9,11.0,0];
        MoveL pTarget,vSpeed,z0,tTool\WObj:=wWobj;
        pTarget.trans:=[12,13.0,0];
        MoveL pTarget,vSpeed,z0,tTool\WObj:=wWobj;
        pTarget.trans:=[18,16.0,0];
        MoveL pTarget,vSpeed,fine,tTool\WObj:=wWobj;
        Reset do_pen;
        MoveL RelTool(pTarget,0,0,-2),vSpeed,z0,tTool\WObj:=wWobj;
        wWobj.oframe.trans.x:=wWobj.oframe.trans.x+16;
    ENDPROC

    ! Character: 0
    PROC char_0()
        VAR robtarget pTarget;
        pTarget:=refTarget;
        pTarget.trans:=[9,32.0,0];
        MoveL pTarget,vSpeed,fine,tTool\WObj:=wWobj;
        Set do_pen;
        pTarget.trans:=[6,31.0,0];
        MoveL pTarget,vSpeed,z0,tTool\WObj:=wWobj;
        pTarget.trans:=[4,28.0,0];
        MoveL pTarget,vSpeed,z0,tTool\WObj:=wWobj;
        pTarget.trans:=[3,23.0,0];
        MoveL pTarget,vSpeed,z0,tTool\WObj:=wWobj;
        pTarget.trans:=[3,20.0,0];
        MoveL pTarget,vSpeed,z0,tTool\WObj:=wWobj;
        pTarget.trans:=[4,15.0,0];
        MoveL pTarget,vSpeed,z0,tTool\WObj:=wWobj;
        pTarget.trans:=[6,12.0,0];
        MoveL pTarget,vSpeed,z0,tTool\WObj:=wWobj;
        pTarget.trans:=[9,11.0,0];
        MoveL pTarget,vSpeed,z0,tTool\WObj:=wWobj;
        pTarget.trans:=[11,11.0,0];
        MoveL pTarget,vSpeed,z0,tTool\WObj:=wWobj;
        pTarget.trans:=[14,12.0,0];
        MoveL pTarget,vSpeed,z0,tTool\WObj:=wWobj;
        pTarget.trans:=[16,15.0,0];
        MoveL pTarget,vSpeed,z0,tTool\WObj:=wWobj;
        pTarget.trans:=[17,20.0,0];
        MoveL pTarget,vSpeed,z0,tTool\WObj:=wWobj;
        pTarget.trans:=[17,23.0,0];
        MoveL pTarget,vSpeed,z0,tTool\WObj:=wWobj;
        pTarget.trans:=[16,28.0,0];
        MoveL pTarget,vSpeed,z0,tTool\WObj:=wWobj;
        pTarget.trans:=[14,31.0,0];
        MoveL pTarget,vSpeed,z0,tTool\WObj:=wWobj;
        pTarget.trans:=[11,32.0,0];
        MoveL pTarget,vSpeed,z0,tTool\WObj:=wWobj;
        pTarget.trans:=[9,32.0,0];
        MoveL pTarget,vSpeed,fine,tTool\WObj:=wWobj;
        Reset do_pen;
        MoveL RelTool(pTarget,0,0,-2),vSpeed,z0,tTool\WObj:=wWobj;
        wWobj.oframe.trans.x:=wWobj.oframe.trans.x+14;
    ENDPROC

    ! Character: 1
    PROC char_1()
        VAR robtarget pTarget;
        pTarget:=refTarget;
        pTarget.trans:=[6,28.0,0];
        MoveL pTarget,vSpeed,fine,tTool\WObj:=wWobj;
        Set do_pen;
        pTarget.trans:=[8,29.0,0];
        MoveL pTarget,vSpeed,z0,tTool\WObj:=wWobj;
        pTarget.trans:=[11,32.0,0];
        MoveL pTarget,vSpeed,z0,tTool\WObj:=wWobj;
        pTarget.trans:=[11,11.0,0];
        MoveL pTarget,vSpeed,fine,tTool\WObj:=wWobj;
        Reset do_pen;
        MoveL RelTool(pTarget,0,0,-2),vSpeed,z0,tTool\WObj:=wWobj;
        wWobj.oframe.trans.x:=wWobj.oframe.trans.x+5;
    ENDPROC

    ! Character: 2
    PROC char_2()
        VAR robtarget pTarget;
        pTarget:=refTarget;
        pTarget.trans:=[4,27.0,0];
        MoveL pTarget,vSpeed,fine,tTool\WObj:=wWobj;
        Set do_pen;
        pTarget.trans:=[4,28.0,0];
        MoveL pTarget,vSpeed,z0,tTool\WObj:=wWobj;
        pTarget.trans:=[5,30.0,0];
        MoveL pTarget,vSpeed,z0,tTool\WObj:=wWobj;
        pTarget.trans:=[6,31.0,0];
        MoveL pTarget,vSpeed,z0,tTool\WObj:=wWobj;
        pTarget.trans:=[8,32.0,0];
        MoveL pTarget,vSpeed,z0,tTool\WObj:=wWobj;
        pTarget.trans:=[12,32.0,0];
        MoveL pTarget,vSpeed,z0,tTool\WObj:=wWobj;
        pTarget.trans:=[14,31.0,0];
        MoveL pTarget,vSpeed,z0,tTool\WObj:=wWobj;
        pTarget.trans:=[15,30.0,0];
        MoveL pTarget,vSpeed,z0,tTool\WObj:=wWobj;
        pTarget.trans:=[16,28.0,0];
        MoveL pTarget,vSpeed,z0,tTool\WObj:=wWobj;
        pTarget.trans:=[16,26.0,0];
        MoveL pTarget,vSpeed,z0,tTool\WObj:=wWobj;
        pTarget.trans:=[15,24.0,0];
        MoveL pTarget,vSpeed,z0,tTool\WObj:=wWobj;
        pTarget.trans:=[13,21.0,0];
        MoveL pTarget,vSpeed,z0,tTool\WObj:=wWobj;
        pTarget.trans:=[3,11.0,0];
        MoveL pTarget,vSpeed,z0,tTool\WObj:=wWobj;
        pTarget.trans:=[17,11.0,0];
        MoveL pTarget,vSpeed,fine,tTool\WObj:=wWobj;
        Reset do_pen;
        MoveL RelTool(pTarget,0,0,-2),vSpeed,z0,tTool\WObj:=wWobj;
        wWobj.oframe.trans.x:=wWobj.oframe.trans.x+14;
    ENDPROC

    ! Character: 3
    PROC char_3()
        VAR robtarget pTarget;
        pTarget:=refTarget;
        pTarget.trans:=[5,32.0,0];
        MoveL pTarget,vSpeed,fine,tTool\WObj:=wWobj;
        Set do_pen;
        pTarget.trans:=[16,32.0,0];
        MoveL pTarget,vSpeed,z0,tTool\WObj:=wWobj;
        pTarget.trans:=[10,24.0,0];
        MoveL pTarget,vSpeed,z0,tTool\WObj:=wWobj;
        pTarget.trans:=[13,24.0,0];
        MoveL pTarget,vSpeed,z0,tTool\WObj:=wWobj;
        pTarget.trans:=[15,23.0,0];
        MoveL pTarget,vSpeed,z0,tTool\WObj:=wWobj;
        pTarget.trans:=[16,22.0,0];
        MoveL pTarget,vSpeed,z0,tTool\WObj:=wWobj;
        pTarget.trans:=[17,19.0,0];
        MoveL pTarget,vSpeed,z0,tTool\WObj:=wWobj;
        pTarget.trans:=[17,17.0,0];
        MoveL pTarget,vSpeed,z0,tTool\WObj:=wWobj;
        pTarget.trans:=[16,14.0,0];
        MoveL pTarget,vSpeed,z0,tTool\WObj:=wWobj;
        pTarget.trans:=[14,12.0,0];
        MoveL pTarget,vSpeed,z0,tTool\WObj:=wWobj;
        pTarget.trans:=[11,11.0,0];
        MoveL pTarget,vSpeed,z0,tTool\WObj:=wWobj;
        pTarget.trans:=[8,11.0,0];
        MoveL pTarget,vSpeed,z0,tTool\WObj:=wWobj;
        pTarget.trans:=[5,12.0,0];
        MoveL pTarget,vSpeed,z0,tTool\WObj:=wWobj;
        pTarget.trans:=[4,13.0,0];
        MoveL pTarget,vSpeed,z0,tTool\WObj:=wWobj;
        pTarget.trans:=[3,15.0,0];
        MoveL pTarget,vSpeed,fine,tTool\WObj:=wWobj;
        Reset do_pen;
        MoveL RelTool(pTarget,0,0,-2),vSpeed,z0,tTool\WObj:=wWobj;
        wWobj.oframe.trans.x:=wWobj.oframe.trans.x+14;
    ENDPROC

    ! Character: 4
    PROC char_4()
        VAR robtarget pTarget;
        pTarget:=refTarget;
        pTarget.trans:=[13,32.0,0];
        MoveL pTarget,vSpeed,fine,tTool\WObj:=wWobj;
        Set do_pen;
        pTarget.trans:=[3,18.0,0];
        MoveL pTarget,vSpeed,z0,tTool\WObj:=wWobj;
        pTarget.trans:=[18,18.0,0];
        MoveL pTarget,vSpeed,fine,tTool\WObj:=wWobj;
        Reset do_pen;
        MoveL RelTool(pTarget,0,0,-2),vSpeed,z0,tTool\WObj:=wWobj;
        pTarget.trans:=[13,32.0,0];
        MoveL pTarget,vSpeed,fine,tTool\WObj:=wWobj;
        Set do_pen;
        pTarget.trans:=[13,11.0,0];
        MoveL pTarget,vSpeed,fine,tTool\WObj:=wWobj;
        Reset do_pen;
        MoveL RelTool(pTarget,0,0,-2),vSpeed,z0,tTool\WObj:=wWobj;
        wWobj.oframe.trans.x:=wWobj.oframe.trans.x+15;
    ENDPROC

    ! Character: 5
    PROC char_5()
        VAR robtarget pTarget;
        pTarget:=refTarget;
        pTarget.trans:=[15,32.0,0];
        MoveL pTarget,vSpeed,fine,tTool\WObj:=wWobj;
        Set do_pen;
        pTarget.trans:=[5,32.0,0];
        MoveL pTarget,vSpeed,z0,tTool\WObj:=wWobj;
        pTarget.trans:=[4,23.0,0];
        MoveL pTarget,vSpeed,z0,tTool\WObj:=wWobj;
        pTarget.trans:=[5,24.0,0];
        MoveL pTarget,vSpeed,z0,tTool\WObj:=wWobj;
        pTarget.trans:=[8,25.0,0];
        MoveL pTarget,vSpeed,z0,tTool\WObj:=wWobj;
        pTarget.trans:=[11,25.0,0];
        MoveL pTarget,vSpeed,z0,tTool\WObj:=wWobj;
        pTarget.trans:=[14,24.0,0];
        MoveL pTarget,vSpeed,z0,tTool\WObj:=wWobj;
        pTarget.trans:=[16,22.0,0];
        MoveL pTarget,vSpeed,z0,tTool\WObj:=wWobj;
        pTarget.trans:=[17,19.0,0];
        MoveL pTarget,vSpeed,z0,tTool\WObj:=wWobj;
        pTarget.trans:=[17,17.0,0];
        MoveL pTarget,vSpeed,z0,tTool\WObj:=wWobj;
        pTarget.trans:=[16,14.0,0];
        MoveL pTarget,vSpeed,z0,tTool\WObj:=wWobj;
        pTarget.trans:=[14,12.0,0];
        MoveL pTarget,vSpeed,z0,tTool\WObj:=wWobj;
        pTarget.trans:=[11,11.0,0];
        MoveL pTarget,vSpeed,z0,tTool\WObj:=wWobj;
        pTarget.trans:=[8,11.0,0];
        MoveL pTarget,vSpeed,z0,tTool\WObj:=wWobj;
        pTarget.trans:=[5,12.0,0];
        MoveL pTarget,vSpeed,z0,tTool\WObj:=wWobj;
        pTarget.trans:=[4,13.0,0];
        MoveL pTarget,vSpeed,z0,tTool\WObj:=wWobj;
        pTarget.trans:=[3,15.0,0];
        MoveL pTarget,vSpeed,fine,tTool\WObj:=wWobj;
        Reset do_pen;
        MoveL RelTool(pTarget,0,0,-2),vSpeed,z0,tTool\WObj:=wWobj;
        wWobj.oframe.trans.x:=wWobj.oframe.trans.x+14;
    ENDPROC

    ! Character: 6
    PROC char_6()
        VAR robtarget pTarget;
        pTarget:=refTarget;
        pTarget.trans:=[16,29.0,0];
        MoveL pTarget,vSpeed,fine,tTool\WObj:=wWobj;
        Set do_pen;
        pTarget.trans:=[15,31.0,0];
        MoveL pTarget,vSpeed,z0,tTool\WObj:=wWobj;
        pTarget.trans:=[12,32.0,0];
        MoveL pTarget,vSpeed,z0,tTool\WObj:=wWobj;
        pTarget.trans:=[10,32.0,0];
        MoveL pTarget,vSpeed,z0,tTool\WObj:=wWobj;
        pTarget.trans:=[7,31.0,0];
        MoveL pTarget,vSpeed,z0,tTool\WObj:=wWobj;
        pTarget.trans:=[5,28.0,0];
        MoveL pTarget,vSpeed,z0,tTool\WObj:=wWobj;
        pTarget.trans:=[4,23.0,0];
        MoveL pTarget,vSpeed,z0,tTool\WObj:=wWobj;
        pTarget.trans:=[4,18.0,0];
        MoveL pTarget,vSpeed,z0,tTool\WObj:=wWobj;
        pTarget.trans:=[5,14.0,0];
        MoveL pTarget,vSpeed,z0,tTool\WObj:=wWobj;
        pTarget.trans:=[7,12.0,0];
        MoveL pTarget,vSpeed,z0,tTool\WObj:=wWobj;
        pTarget.trans:=[10,11.0,0];
        MoveL pTarget,vSpeed,z0,tTool\WObj:=wWobj;
        pTarget.trans:=[11,11.0,0];
        MoveL pTarget,vSpeed,z0,tTool\WObj:=wWobj;
        pTarget.trans:=[14,12.0,0];
        MoveL pTarget,vSpeed,z0,tTool\WObj:=wWobj;
        pTarget.trans:=[16,14.0,0];
        MoveL pTarget,vSpeed,z0,tTool\WObj:=wWobj;
        pTarget.trans:=[17,17.0,0];
        MoveL pTarget,vSpeed,z0,tTool\WObj:=wWobj;
        pTarget.trans:=[17,18.0,0];
        MoveL pTarget,vSpeed,z0,tTool\WObj:=wWobj;
        pTarget.trans:=[16,21.0,0];
        MoveL pTarget,vSpeed,z0,tTool\WObj:=wWobj;
        pTarget.trans:=[14,23.0,0];
        MoveL pTarget,vSpeed,z0,tTool\WObj:=wWobj;
        pTarget.trans:=[11,24.0,0];
        MoveL pTarget,vSpeed,z0,tTool\WObj:=wWobj;
        pTarget.trans:=[10,24.0,0];
        MoveL pTarget,vSpeed,z0,tTool\WObj:=wWobj;
        pTarget.trans:=[7,23.0,0];
        MoveL pTarget,vSpeed,z0,tTool\WObj:=wWobj;
        pTarget.trans:=[5,21.0,0];
        MoveL pTarget,vSpeed,z0,tTool\WObj:=wWobj;
        pTarget.trans:=[4,18.0,0];
        MoveL pTarget,vSpeed,fine,tTool\WObj:=wWobj;
        Reset do_pen;
        MoveL RelTool(pTarget,0,0,-2),vSpeed,z0,tTool\WObj:=wWobj;
        wWobj.oframe.trans.x:=wWobj.oframe.trans.x+13;
    ENDPROC

    ! Character: 7
    PROC char_7()
        VAR robtarget pTarget;
        pTarget:=refTarget;
        pTarget.trans:=[17,32.0,0];
        MoveL pTarget,vSpeed,fine,tTool\WObj:=wWobj;
        Set do_pen;
        pTarget.trans:=[7,11.0,0];
        MoveL pTarget,vSpeed,fine,tTool\WObj:=wWobj;
        Reset do_pen;
        MoveL RelTool(pTarget,0,0,-2),vSpeed,z0,tTool\WObj:=wWobj;
        pTarget.trans:=[3,32.0,0];
        MoveL pTarget,vSpeed,fine,tTool\WObj:=wWobj;
        Set do_pen;
        pTarget.trans:=[17,32.0,0];
        MoveL pTarget,vSpeed,fine,tTool\WObj:=wWobj;
        Reset do_pen;
        MoveL RelTool(pTarget,0,0,-2),vSpeed,z0,tTool\WObj:=wWobj;
        wWobj.oframe.trans.x:=wWobj.oframe.trans.x+14;
    ENDPROC

    ! Character: 8
    PROC char_8()
        VAR robtarget pTarget;
        pTarget:=refTarget;
        pTarget.trans:=[8,32.0,0];
        MoveL pTarget,vSpeed,fine,tTool\WObj:=wWobj;
        Set do_pen;
        pTarget.trans:=[5,31.0,0];
        MoveL pTarget,vSpeed,z0,tTool\WObj:=wWobj;
        pTarget.trans:=[4,29.0,0];
        MoveL pTarget,vSpeed,z0,tTool\WObj:=wWobj;
        pTarget.trans:=[4,27.0,0];
        MoveL pTarget,vSpeed,z0,tTool\WObj:=wWobj;
        pTarget.trans:=[5,25.0,0];
        MoveL pTarget,vSpeed,z0,tTool\WObj:=wWobj;
        pTarget.trans:=[7,24.0,0];
        MoveL pTarget,vSpeed,z0,tTool\WObj:=wWobj;
        pTarget.trans:=[11,23.0,0];
        MoveL pTarget,vSpeed,z0,tTool\WObj:=wWobj;
        pTarget.trans:=[14,22.0,0];
        MoveL pTarget,vSpeed,z0,tTool\WObj:=wWobj;
        pTarget.trans:=[16,20.0,0];
        MoveL pTarget,vSpeed,z0,tTool\WObj:=wWobj;
        pTarget.trans:=[17,18.0,0];
        MoveL pTarget,vSpeed,z0,tTool\WObj:=wWobj;
        pTarget.trans:=[17,15.0,0];
        MoveL pTarget,vSpeed,z0,tTool\WObj:=wWobj;
        pTarget.trans:=[16,13.0,0];
        MoveL pTarget,vSpeed,z0,tTool\WObj:=wWobj;
        pTarget.trans:=[15,12.0,0];
        MoveL pTarget,vSpeed,z0,tTool\WObj:=wWobj;
        pTarget.trans:=[12,11.0,0];
        MoveL pTarget,vSpeed,z0,tTool\WObj:=wWobj;
        pTarget.trans:=[8,11.0,0];
        MoveL pTarget,vSpeed,z0,tTool\WObj:=wWobj;
        pTarget.trans:=[5,12.0,0];
        MoveL pTarget,vSpeed,z0,tTool\WObj:=wWobj;
        pTarget.trans:=[4,13.0,0];
        MoveL pTarget,vSpeed,z0,tTool\WObj:=wWobj;
        pTarget.trans:=[3,15.0,0];
        MoveL pTarget,vSpeed,z0,tTool\WObj:=wWobj;
        pTarget.trans:=[3,18.0,0];
        MoveL pTarget,vSpeed,z0,tTool\WObj:=wWobj;
        pTarget.trans:=[4,20.0,0];
        MoveL pTarget,vSpeed,z0,tTool\WObj:=wWobj;
        pTarget.trans:=[6,22.0,0];
        MoveL pTarget,vSpeed,z0,tTool\WObj:=wWobj;
        pTarget.trans:=[9,23.0,0];
        MoveL pTarget,vSpeed,z0,tTool\WObj:=wWobj;
        pTarget.trans:=[13,24.0,0];
        MoveL pTarget,vSpeed,z0,tTool\WObj:=wWobj;
        pTarget.trans:=[15,25.0,0];
        MoveL pTarget,vSpeed,z0,tTool\WObj:=wWobj;
        pTarget.trans:=[16,27.0,0];
        MoveL pTarget,vSpeed,z0,tTool\WObj:=wWobj;
        pTarget.trans:=[16,29.0,0];
        MoveL pTarget,vSpeed,z0,tTool\WObj:=wWobj;
        pTarget.trans:=[15,31.0,0];
        MoveL pTarget,vSpeed,z0,tTool\WObj:=wWobj;
        pTarget.trans:=[12,32.0,0];
        MoveL pTarget,vSpeed,z0,tTool\WObj:=wWobj;
        pTarget.trans:=[8,32.0,0];
        MoveL pTarget,vSpeed,fine,tTool\WObj:=wWobj;
        Reset do_pen;
        MoveL RelTool(pTarget,0,0,-2),vSpeed,z0,tTool\WObj:=wWobj;
        wWobj.oframe.trans.x:=wWobj.oframe.trans.x+14;
    ENDPROC

    ! Character: 9
    PROC char_9()
        VAR robtarget pTarget;
        pTarget:=refTarget;
        pTarget.trans:=[16,25.0,0];
        MoveL pTarget,vSpeed,fine,tTool\WObj:=wWobj;
        Set do_pen;
        pTarget.trans:=[15,22.0,0];
        MoveL pTarget,vSpeed,z0,tTool\WObj:=wWobj;
        pTarget.trans:=[13,20.0,0];
        MoveL pTarget,vSpeed,z0,tTool\WObj:=wWobj;
        pTarget.trans:=[10,19.0,0];
        MoveL pTarget,vSpeed,z0,tTool\WObj:=wWobj;
        pTarget.trans:=[9,19.0,0];
        MoveL pTarget,vSpeed,z0,tTool\WObj:=wWobj;
        pTarget.trans:=[6,20.0,0];
        MoveL pTarget,vSpeed,z0,tTool\WObj:=wWobj;
        pTarget.trans:=[4,22.0,0];
        MoveL pTarget,vSpeed,z0,tTool\WObj:=wWobj;
        pTarget.trans:=[3,25.0,0];
        MoveL pTarget,vSpeed,z0,tTool\WObj:=wWobj;
        pTarget.trans:=[3,26.0,0];
        MoveL pTarget,vSpeed,z0,tTool\WObj:=wWobj;
        pTarget.trans:=[4,29.0,0];
        MoveL pTarget,vSpeed,z0,tTool\WObj:=wWobj;
        pTarget.trans:=[6,31.0,0];
        MoveL pTarget,vSpeed,z0,tTool\WObj:=wWobj;
        pTarget.trans:=[9,32.0,0];
        MoveL pTarget,vSpeed,z0,tTool\WObj:=wWobj;
        pTarget.trans:=[10,32.0,0];
        MoveL pTarget,vSpeed,z0,tTool\WObj:=wWobj;
        pTarget.trans:=[13,31.0,0];
        MoveL pTarget,vSpeed,z0,tTool\WObj:=wWobj;
        pTarget.trans:=[15,29.0,0];
        MoveL pTarget,vSpeed,z0,tTool\WObj:=wWobj;
        pTarget.trans:=[16,25.0,0];
        MoveL pTarget,vSpeed,z0,tTool\WObj:=wWobj;
        pTarget.trans:=[16,20.0,0];
        MoveL pTarget,vSpeed,z0,tTool\WObj:=wWobj;
        pTarget.trans:=[15,15.0,0];
        MoveL pTarget,vSpeed,z0,tTool\WObj:=wWobj;
        pTarget.trans:=[13,12.0,0];
        MoveL pTarget,vSpeed,z0,tTool\WObj:=wWobj;
        pTarget.trans:=[10,11.0,0];
        MoveL pTarget,vSpeed,z0,tTool\WObj:=wWobj;
        pTarget.trans:=[8,11.0,0];
        MoveL pTarget,vSpeed,z0,tTool\WObj:=wWobj;
        pTarget.trans:=[5,12.0,0];
        MoveL pTarget,vSpeed,z0,tTool\WObj:=wWobj;
        pTarget.trans:=[4,14.0,0];
        MoveL pTarget,vSpeed,fine,tTool\WObj:=wWobj;
        Reset do_pen;
        MoveL RelTool(pTarget,0,0,-2),vSpeed,z0,tTool\WObj:=wWobj;
        wWobj.oframe.trans.x:=wWobj.oframe.trans.x+13;
    ENDPROC

    ! Character: !
    PROC char_exclamation()
        VAR robtarget pTarget;
        pTarget:=refTarget;
        pTarget.trans:=[5,32.0,0];
        MoveL pTarget,vSpeed,fine,tTool\WObj:=wWobj;
        Set do_pen;
        pTarget.trans:=[5,18.0,0];
        MoveL pTarget,vSpeed,fine,tTool\WObj:=wWobj;
        Reset do_pen;
        MoveL RelTool(pTarget,0,0,-2),vSpeed,z0,tTool\WObj:=wWobj;
        pTarget.trans:=[5,13.0,0];
        MoveL pTarget,vSpeed,fine,tTool\WObj:=wWobj;
        Set do_pen;
        pTarget.trans:=[4,12.0,0];
        MoveL pTarget,vSpeed,z0,tTool\WObj:=wWobj;
        pTarget.trans:=[5,11.0,0];
        MoveL pTarget,vSpeed,z0,tTool\WObj:=wWobj;
        pTarget.trans:=[6,12.0,0];
        MoveL pTarget,vSpeed,z0,tTool\WObj:=wWobj;
        pTarget.trans:=[5,13.0,0];
        MoveL pTarget,vSpeed,fine,tTool\WObj:=wWobj;
        Reset do_pen;
        MoveL RelTool(pTarget,0,0,-2),vSpeed,z0,tTool\WObj:=wWobj;
        wWobj.oframe.trans.x:=wWobj.oframe.trans.x+2;
    ENDPROC

    ! Character: @
    PROC char_at()
        VAR robtarget pTarget;
        pTarget:=refTarget;
        pTarget.trans:=[18,24.0,0];
        MoveL pTarget,vSpeed,fine,tTool\WObj:=wWobj;
        Set do_pen;
        pTarget.trans:=[17,26.0,0];
        MoveL pTarget,vSpeed,z0,tTool\WObj:=wWobj;
        pTarget.trans:=[15,27.0,0];
        MoveL pTarget,vSpeed,z0,tTool\WObj:=wWobj;
        pTarget.trans:=[12,27.0,0];
        MoveL pTarget,vSpeed,z0,tTool\WObj:=wWobj;
        pTarget.trans:=[10,26.0,0];
        MoveL pTarget,vSpeed,z0,tTool\WObj:=wWobj;
        pTarget.trans:=[9,25.0,0];
        MoveL pTarget,vSpeed,z0,tTool\WObj:=wWobj;
        pTarget.trans:=[8,22.0,0];
        MoveL pTarget,vSpeed,z0,tTool\WObj:=wWobj;
        pTarget.trans:=[8,19.0,0];
        MoveL pTarget,vSpeed,z0,tTool\WObj:=wWobj;
        pTarget.trans:=[9,17.0,0];
        MoveL pTarget,vSpeed,z0,tTool\WObj:=wWobj;
        pTarget.trans:=[11,16.0,0];
        MoveL pTarget,vSpeed,z0,tTool\WObj:=wWobj;
        pTarget.trans:=[14,16.0,0];
        MoveL pTarget,vSpeed,z0,tTool\WObj:=wWobj;
        pTarget.trans:=[16,17.0,0];
        MoveL pTarget,vSpeed,z0,tTool\WObj:=wWobj;
        pTarget.trans:=[17,19.0,0];
        MoveL pTarget,vSpeed,fine,tTool\WObj:=wWobj;
        Reset do_pen;
        MoveL RelTool(pTarget,0,0,-2),vSpeed,z0,tTool\WObj:=wWobj;
        pTarget.trans:=[12,27.0,0];
        MoveL pTarget,vSpeed,fine,tTool\WObj:=wWobj;
        Set do_pen;
        pTarget.trans:=[10,25.0,0];
        MoveL pTarget,vSpeed,z0,tTool\WObj:=wWobj;
        pTarget.trans:=[9,22.0,0];
        MoveL pTarget,vSpeed,z0,tTool\WObj:=wWobj;
        pTarget.trans:=[9,19.0,0];
        MoveL pTarget,vSpeed,z0,tTool\WObj:=wWobj;
        pTarget.trans:=[10,17.0,0];
        MoveL pTarget,vSpeed,z0,tTool\WObj:=wWobj;
        pTarget.trans:=[11,16.0,0];
        MoveL pTarget,vSpeed,fine,tTool\WObj:=wWobj;
        Reset do_pen;
        MoveL RelTool(pTarget,0,0,-2),vSpeed,z0,tTool\WObj:=wWobj;
        pTarget.trans:=[18,27.0,0];
        MoveL pTarget,vSpeed,fine,tTool\WObj:=wWobj;
        Set do_pen;
        pTarget.trans:=[17,19.0,0];
        MoveL pTarget,vSpeed,z0,tTool\WObj:=wWobj;
        pTarget.trans:=[17,17.0,0];
        MoveL pTarget,vSpeed,z0,tTool\WObj:=wWobj;
        pTarget.trans:=[19,16.0,0];
        MoveL pTarget,vSpeed,z0,tTool\WObj:=wWobj;
        pTarget.trans:=[21,16.0,0];
        MoveL pTarget,vSpeed,z0,tTool\WObj:=wWobj;
        pTarget.trans:=[23,18.0,0];
        MoveL pTarget,vSpeed,z0,tTool\WObj:=wWobj;
        pTarget.trans:=[24,21.0,0];
        MoveL pTarget,vSpeed,z0,tTool\WObj:=wWobj;
        pTarget.trans:=[24,23.0,0];
        MoveL pTarget,vSpeed,z0,tTool\WObj:=wWobj;
        pTarget.trans:=[23,26.0,0];
        MoveL pTarget,vSpeed,z0,tTool\WObj:=wWobj;
        pTarget.trans:=[22,28.0,0];
        MoveL pTarget,vSpeed,z0,tTool\WObj:=wWobj;
        pTarget.trans:=[20,30.0,0];
        MoveL pTarget,vSpeed,z0,tTool\WObj:=wWobj;
        pTarget.trans:=[18,31.0,0];
        MoveL pTarget,vSpeed,z0,tTool\WObj:=wWobj;
        pTarget.trans:=[15,32.0,0];
        MoveL pTarget,vSpeed,z0,tTool\WObj:=wWobj;
        pTarget.trans:=[12,32.0,0];
        MoveL pTarget,vSpeed,z0,tTool\WObj:=wWobj;
        pTarget.trans:=[9,31.0,0];
        MoveL pTarget,vSpeed,z0,tTool\WObj:=wWobj;
        pTarget.trans:=[7,30.0,0];
        MoveL pTarget,vSpeed,z0,tTool\WObj:=wWobj;
        pTarget.trans:=[5,28.0,0];
        MoveL pTarget,vSpeed,z0,tTool\WObj:=wWobj;
        pTarget.trans:=[4,26.0,0];
        MoveL pTarget,vSpeed,z0,tTool\WObj:=wWobj;
        pTarget.trans:=[3,23.0,0];
        MoveL pTarget,vSpeed,z0,tTool\WObj:=wWobj;
        pTarget.trans:=[3,20.0,0];
        MoveL pTarget,vSpeed,z0,tTool\WObj:=wWobj;
        pTarget.trans:=[4,17.0,0];
        MoveL pTarget,vSpeed,z0,tTool\WObj:=wWobj;
        pTarget.trans:=[5,15.0,0];
        MoveL pTarget,vSpeed,z0,tTool\WObj:=wWobj;
        pTarget.trans:=[7,13.0,0];
        MoveL pTarget,vSpeed,z0,tTool\WObj:=wWobj;
        pTarget.trans:=[9,12.0,0];
        MoveL pTarget,vSpeed,z0,tTool\WObj:=wWobj;
        pTarget.trans:=[12,11.0,0];
        MoveL pTarget,vSpeed,z0,tTool\WObj:=wWobj;
        pTarget.trans:=[15,11.0,0];
        MoveL pTarget,vSpeed,z0,tTool\WObj:=wWobj;
        pTarget.trans:=[18,12.0,0];
        MoveL pTarget,vSpeed,z0,tTool\WObj:=wWobj;
        pTarget.trans:=[20,13.0,0];
        MoveL pTarget,vSpeed,z0,tTool\WObj:=wWobj;
        pTarget.trans:=[21,14.0,0];
        MoveL pTarget,vSpeed,fine,tTool\WObj:=wWobj;
        Reset do_pen;
        MoveL RelTool(pTarget,0,0,-2),vSpeed,z0,tTool\WObj:=wWobj;
        pTarget.trans:=[19,27.0,0];
        MoveL pTarget,vSpeed,fine,tTool\WObj:=wWobj;
        Set do_pen;
        pTarget.trans:=[18,19.0,0];
        MoveL pTarget,vSpeed,z0,tTool\WObj:=wWobj;
        pTarget.trans:=[18,17.0,0];
        MoveL pTarget,vSpeed,z0,tTool\WObj:=wWobj;
        pTarget.trans:=[19,16.0,0];
        MoveL pTarget,vSpeed,fine,tTool\WObj:=wWobj;
        Reset do_pen;
        MoveL RelTool(pTarget,0,0,-2),vSpeed,z0,tTool\WObj:=wWobj;
        wWobj.oframe.trans.x:=wWobj.oframe.trans.x+21;
    ENDPROC

    ! Character: #
    PROC char_hash()
        VAR robtarget pTarget;
        pTarget:=refTarget;
        pTarget.trans:=[11,36.0,0];
        MoveL pTarget,vSpeed,fine,tTool\WObj:=wWobj;
        Set do_pen;
        pTarget.trans:=[4,4.0,0];
        MoveL pTarget,vSpeed,fine,tTool\WObj:=wWobj;
        Reset do_pen;
        MoveL RelTool(pTarget,0,0,-2),vSpeed,z0,tTool\WObj:=wWobj;
        pTarget.trans:=[17,36.0,0];
        MoveL pTarget,vSpeed,fine,tTool\WObj:=wWobj;
        Set do_pen;
        pTarget.trans:=[10,4.0,0];
        MoveL pTarget,vSpeed,fine,tTool\WObj:=wWobj;
        Reset do_pen;
        MoveL RelTool(pTarget,0,0,-2),vSpeed,z0,tTool\WObj:=wWobj;
        pTarget.trans:=[4,23.0,0];
        MoveL pTarget,vSpeed,fine,tTool\WObj:=wWobj;
        Set do_pen;
        pTarget.trans:=[18,23.0,0];
        MoveL pTarget,vSpeed,fine,tTool\WObj:=wWobj;
        Reset do_pen;
        MoveL RelTool(pTarget,0,0,-2),vSpeed,z0,tTool\WObj:=wWobj;
        pTarget.trans:=[3,17.0,0];
        MoveL pTarget,vSpeed,fine,tTool\WObj:=wWobj;
        Set do_pen;
        pTarget.trans:=[17,17.0,0];
        MoveL pTarget,vSpeed,fine,tTool\WObj:=wWobj;
        Reset do_pen;
        MoveL RelTool(pTarget,0,0,-2),vSpeed,z0,tTool\WObj:=wWobj;
        wWobj.oframe.trans.x:=wWobj.oframe.trans.x+15;
    ENDPROC

    ! Character: $
    PROC char_dollar()
        VAR robtarget pTarget;
        pTarget:=refTarget;
        pTarget.trans:=[8,36.0,0];
        MoveL pTarget,vSpeed,fine,tTool\WObj:=wWobj;
        Set do_pen;
        pTarget.trans:=[8,7.0,0];
        MoveL pTarget,vSpeed,fine,tTool\WObj:=wWobj;
        Reset do_pen;
        MoveL RelTool(pTarget,0,0,-2),vSpeed,z0,tTool\WObj:=wWobj;
        pTarget.trans:=[12,36.0,0];
        MoveL pTarget,vSpeed,fine,tTool\WObj:=wWobj;
        Set do_pen;
        pTarget.trans:=[12,7.0,0];
        MoveL pTarget,vSpeed,fine,tTool\WObj:=wWobj;
        Reset do_pen;
        MoveL RelTool(pTarget,0,0,-2),vSpeed,z0,tTool\WObj:=wWobj;
        pTarget.trans:=[17,29.0,0];
        MoveL pTarget,vSpeed,fine,tTool\WObj:=wWobj;
        Set do_pen;
        pTarget.trans:=[15,31.0,0];
        MoveL pTarget,vSpeed,z0,tTool\WObj:=wWobj;
        pTarget.trans:=[12,32.0,0];
        MoveL pTarget,vSpeed,z0,tTool\WObj:=wWobj;
        pTarget.trans:=[8,32.0,0];
        MoveL pTarget,vSpeed,z0,tTool\WObj:=wWobj;
        pTarget.trans:=[5,31.0,0];
        MoveL pTarget,vSpeed,z0,tTool\WObj:=wWobj;
        pTarget.trans:=[3,29.0,0];
        MoveL pTarget,vSpeed,z0,tTool\WObj:=wWobj;
        pTarget.trans:=[3,27.0,0];
        MoveL pTarget,vSpeed,z0,tTool\WObj:=wWobj;
        pTarget.trans:=[4,25.0,0];
        MoveL pTarget,vSpeed,z0,tTool\WObj:=wWobj;
        pTarget.trans:=[5,24.0,0];
        MoveL pTarget,vSpeed,z0,tTool\WObj:=wWobj;
        pTarget.trans:=[7,23.0,0];
        MoveL pTarget,vSpeed,z0,tTool\WObj:=wWobj;
        pTarget.trans:=[13,21.0,0];
        MoveL pTarget,vSpeed,z0,tTool\WObj:=wWobj;
        pTarget.trans:=[15,20.0,0];
        MoveL pTarget,vSpeed,z0,tTool\WObj:=wWobj;
        pTarget.trans:=[16,19.0,0];
        MoveL pTarget,vSpeed,z0,tTool\WObj:=wWobj;
        pTarget.trans:=[17,17.0,0];
        MoveL pTarget,vSpeed,z0,tTool\WObj:=wWobj;
        pTarget.trans:=[17,14.0,0];
        MoveL pTarget,vSpeed,z0,tTool\WObj:=wWobj;
        pTarget.trans:=[15,12.0,0];
        MoveL pTarget,vSpeed,z0,tTool\WObj:=wWobj;
        pTarget.trans:=[12,11.0,0];
        MoveL pTarget,vSpeed,z0,tTool\WObj:=wWobj;
        pTarget.trans:=[8,11.0,0];
        MoveL pTarget,vSpeed,z0,tTool\WObj:=wWobj;
        pTarget.trans:=[5,12.0,0];
        MoveL pTarget,vSpeed,z0,tTool\WObj:=wWobj;
        pTarget.trans:=[3,14.0,0];
        MoveL pTarget,vSpeed,fine,tTool\WObj:=wWobj;
        Reset do_pen;
        MoveL RelTool(pTarget,0,0,-2),vSpeed,z0,tTool\WObj:=wWobj;
        wWobj.oframe.trans.x:=wWobj.oframe.trans.x+14;
    ENDPROC

    ! Character: %
    PROC char_percent()
        VAR robtarget pTarget;
        pTarget:=refTarget;
        pTarget.trans:=[21,32.0,0];
        MoveL pTarget,vSpeed,fine,tTool\WObj:=wWobj;
        Set do_pen;
        pTarget.trans:=[3,11.0,0];
        MoveL pTarget,vSpeed,fine,tTool\WObj:=wWobj;
        Reset do_pen;
        MoveL RelTool(pTarget,0,0,-2),vSpeed,z0,tTool\WObj:=wWobj;
        pTarget.trans:=[8,32.0,0];
        MoveL pTarget,vSpeed,fine,tTool\WObj:=wWobj;
        Set do_pen;
        pTarget.trans:=[10,30.0,0];
        MoveL pTarget,vSpeed,z0,tTool\WObj:=wWobj;
        pTarget.trans:=[10,28.0,0];
        MoveL pTarget,vSpeed,z0,tTool\WObj:=wWobj;
        pTarget.trans:=[9,26.0,0];
        MoveL pTarget,vSpeed,z0,tTool\WObj:=wWobj;
        pTarget.trans:=[7,25.0,0];
        MoveL pTarget,vSpeed,z0,tTool\WObj:=wWobj;
        pTarget.trans:=[5,25.0,0];
        MoveL pTarget,vSpeed,z0,tTool\WObj:=wWobj;
        pTarget.trans:=[3,27.0,0];
        MoveL pTarget,vSpeed,z0,tTool\WObj:=wWobj;
        pTarget.trans:=[3,29.0,0];
        MoveL pTarget,vSpeed,z0,tTool\WObj:=wWobj;
        pTarget.trans:=[4,31.0,0];
        MoveL pTarget,vSpeed,z0,tTool\WObj:=wWobj;
        pTarget.trans:=[6,32.0,0];
        MoveL pTarget,vSpeed,z0,tTool\WObj:=wWobj;
        pTarget.trans:=[8,32.0,0];
        MoveL pTarget,vSpeed,z0,tTool\WObj:=wWobj;
        pTarget.trans:=[10,31.0,0];
        MoveL pTarget,vSpeed,z0,tTool\WObj:=wWobj;
        pTarget.trans:=[13,30.0,0];
        MoveL pTarget,vSpeed,z0,tTool\WObj:=wWobj;
        pTarget.trans:=[16,30.0,0];
        MoveL pTarget,vSpeed,z0,tTool\WObj:=wWobj;
        pTarget.trans:=[19,31.0,0];
        MoveL pTarget,vSpeed,z0,tTool\WObj:=wWobj;
        pTarget.trans:=[21,32.0,0];
        MoveL pTarget,vSpeed,fine,tTool\WObj:=wWobj;
        Reset do_pen;
        MoveL RelTool(pTarget,0,0,-2),vSpeed,z0,tTool\WObj:=wWobj;
        pTarget.trans:=[17,18.0,0];
        MoveL pTarget,vSpeed,fine,tTool\WObj:=wWobj;
        Set do_pen;
        pTarget.trans:=[15,17.0,0];
        MoveL pTarget,vSpeed,z0,tTool\WObj:=wWobj;
        pTarget.trans:=[14,15.0,0];
        MoveL pTarget,vSpeed,z0,tTool\WObj:=wWobj;
        pTarget.trans:=[14,13.0,0];
        MoveL pTarget,vSpeed,z0,tTool\WObj:=wWobj;
        pTarget.trans:=[16,11.0,0];
        MoveL pTarget,vSpeed,z0,tTool\WObj:=wWobj;
        pTarget.trans:=[18,11.0,0];
        MoveL pTarget,vSpeed,z0,tTool\WObj:=wWobj;
        pTarget.trans:=[20,12.0,0];
        MoveL pTarget,vSpeed,z0,tTool\WObj:=wWobj;
        pTarget.trans:=[21,14.0,0];
        MoveL pTarget,vSpeed,z0,tTool\WObj:=wWobj;
        pTarget.trans:=[21,16.0,0];
        MoveL pTarget,vSpeed,z0,tTool\WObj:=wWobj;
        pTarget.trans:=[19,18.0,0];
        MoveL pTarget,vSpeed,z0,tTool\WObj:=wWobj;
        pTarget.trans:=[17,18.0,0];
        MoveL pTarget,vSpeed,fine,tTool\WObj:=wWobj;
        Reset do_pen;
        MoveL RelTool(pTarget,0,0,-2),vSpeed,z0,tTool\WObj:=wWobj;
        wWobj.oframe.trans.x:=wWobj.oframe.trans.x+18;
    ENDPROC

    ! Character: ^
    PROC char_caret()
        VAR robtarget pTarget;
        pTarget:=refTarget;
        pTarget.trans:=[8,34.0,0];
        MoveL pTarget,vSpeed,fine,tTool\WObj:=wWobj;
        Set do_pen;
        pTarget.trans:=[0,20.0,0];
        MoveL pTarget,vSpeed,fine,tTool\WObj:=wWobj;
        Reset do_pen;
        MoveL RelTool(pTarget,0,0,-2),vSpeed,z0,tTool\WObj:=wWobj;
        pTarget.trans:=[8,34.0,0];
        MoveL pTarget,vSpeed,fine,tTool\WObj:=wWobj;
        Set do_pen;
        pTarget.trans:=[16,20.0,0];
        MoveL pTarget,vSpeed,fine,tTool\WObj:=wWobj;
        Reset do_pen;
        MoveL RelTool(pTarget,0,0,-2),vSpeed,z0,tTool\WObj:=wWobj;
        wWobj.oframe.trans.x:=wWobj.oframe.trans.x+16;
    ENDPROC

    ! Character: &
    PROC char_ampersand()
        VAR robtarget pTarget;
        pTarget:=refTarget;
        pTarget.trans:=[23,23.0,0];
        MoveL pTarget,vSpeed,fine,tTool\WObj:=wWobj;
        Set do_pen;
        pTarget.trans:=[23,24.0,0];
        MoveL pTarget,vSpeed,z0,tTool\WObj:=wWobj;
        pTarget.trans:=[22,25.0,0];
        MoveL pTarget,vSpeed,z0,tTool\WObj:=wWobj;
        pTarget.trans:=[21,25.0,0];
        MoveL pTarget,vSpeed,z0,tTool\WObj:=wWobj;
        pTarget.trans:=[20,24.0,0];
        MoveL pTarget,vSpeed,z0,tTool\WObj:=wWobj;
        pTarget.trans:=[19,22.0,0];
        MoveL pTarget,vSpeed,z0,tTool\WObj:=wWobj;
        pTarget.trans:=[17,17.0,0];
        MoveL pTarget,vSpeed,z0,tTool\WObj:=wWobj;
        pTarget.trans:=[15,14.0,0];
        MoveL pTarget,vSpeed,z0,tTool\WObj:=wWobj;
        pTarget.trans:=[13,12.0,0];
        MoveL pTarget,vSpeed,z0,tTool\WObj:=wWobj;
        pTarget.trans:=[11,11.0,0];
        MoveL pTarget,vSpeed,z0,tTool\WObj:=wWobj;
        pTarget.trans:=[7,11.0,0];
        MoveL pTarget,vSpeed,z0,tTool\WObj:=wWobj;
        pTarget.trans:=[5,12.0,0];
        MoveL pTarget,vSpeed,z0,tTool\WObj:=wWobj;
        pTarget.trans:=[4,13.0,0];
        MoveL pTarget,vSpeed,z0,tTool\WObj:=wWobj;
        pTarget.trans:=[3,15.0,0];
        MoveL pTarget,vSpeed,z0,tTool\WObj:=wWobj;
        pTarget.trans:=[3,17.0,0];
        MoveL pTarget,vSpeed,z0,tTool\WObj:=wWobj;
        pTarget.trans:=[4,19.0,0];
        MoveL pTarget,vSpeed,z0,tTool\WObj:=wWobj;
        pTarget.trans:=[5,20.0,0];
        MoveL pTarget,vSpeed,z0,tTool\WObj:=wWobj;
        pTarget.trans:=[12,24.0,0];
        MoveL pTarget,vSpeed,z0,tTool\WObj:=wWobj;
        pTarget.trans:=[13,25.0,0];
        MoveL pTarget,vSpeed,z0,tTool\WObj:=wWobj;
        pTarget.trans:=[14,27.0,0];
        MoveL pTarget,vSpeed,z0,tTool\WObj:=wWobj;
        pTarget.trans:=[14,29.0,0];
        MoveL pTarget,vSpeed,z0,tTool\WObj:=wWobj;
        pTarget.trans:=[13,31.0,0];
        MoveL pTarget,vSpeed,z0,tTool\WObj:=wWobj;
        pTarget.trans:=[11,32.0,0];
        MoveL pTarget,vSpeed,z0,tTool\WObj:=wWobj;
        pTarget.trans:=[9,31.0,0];
        MoveL pTarget,vSpeed,z0,tTool\WObj:=wWobj;
        pTarget.trans:=[8,29.0,0];
        MoveL pTarget,vSpeed,z0,tTool\WObj:=wWobj;
        pTarget.trans:=[8,27.0,0];
        MoveL pTarget,vSpeed,z0,tTool\WObj:=wWobj;
        pTarget.trans:=[9,24.0,0];
        MoveL pTarget,vSpeed,z0,tTool\WObj:=wWobj;
        pTarget.trans:=[11,21.0,0];
        MoveL pTarget,vSpeed,z0,tTool\WObj:=wWobj;
        pTarget.trans:=[16,14.0,0];
        MoveL pTarget,vSpeed,z0,tTool\WObj:=wWobj;
        pTarget.trans:=[18,12.0,0];
        MoveL pTarget,vSpeed,z0,tTool\WObj:=wWobj;
        pTarget.trans:=[20,11.0,0];
        MoveL pTarget,vSpeed,z0,tTool\WObj:=wWobj;
        pTarget.trans:=[22,11.0,0];
        MoveL pTarget,vSpeed,z0,tTool\WObj:=wWobj;
        pTarget.trans:=[23,12.0,0];
        MoveL pTarget,vSpeed,z0,tTool\WObj:=wWobj;
        pTarget.trans:=[23,13.0,0];
        MoveL pTarget,vSpeed,fine,tTool\WObj:=wWobj;
        Reset do_pen;
        MoveL RelTool(pTarget,0,0,-2),vSpeed,z0,tTool\WObj:=wWobj;
        wWobj.oframe.trans.x:=wWobj.oframe.trans.x+20;
    ENDPROC

    ! Character: *
    PROC char_asterisk()
        VAR robtarget pTarget;
        pTarget:=refTarget;
        pTarget.trans:=[8,26.0,0];
        MoveL pTarget,vSpeed,fine,tTool\WObj:=wWobj;
        Set do_pen;
        pTarget.trans:=[8,14.0,0];
        MoveL pTarget,vSpeed,fine,tTool\WObj:=wWobj;
        Reset do_pen;
        MoveL RelTool(pTarget,0,0,-2),vSpeed,z0,tTool\WObj:=wWobj;
        pTarget.trans:=[3,23.0,0];
        MoveL pTarget,vSpeed,fine,tTool\WObj:=wWobj;
        Set do_pen;
        pTarget.trans:=[13,17.0,0];
        MoveL pTarget,vSpeed,fine,tTool\WObj:=wWobj;
        Reset do_pen;
        MoveL RelTool(pTarget,0,0,-2),vSpeed,z0,tTool\WObj:=wWobj;
        pTarget.trans:=[13,23.0,0];
        MoveL pTarget,vSpeed,fine,tTool\WObj:=wWobj;
        Set do_pen;
        pTarget.trans:=[3,17.0,0];
        MoveL pTarget,vSpeed,fine,tTool\WObj:=wWobj;
        Reset do_pen;
        MoveL RelTool(pTarget,0,0,-2),vSpeed,z0,tTool\WObj:=wWobj;
        wWobj.oframe.trans.x:=wWobj.oframe.trans.x+10;
    ENDPROC

    ! Character: (
    PROC char_leftparenthesis()
        VAR robtarget pTarget;
        pTarget:=refTarget;
        pTarget.trans:=[11,36.0,0];
        MoveL pTarget,vSpeed,fine,tTool\WObj:=wWobj;
        Set do_pen;
        pTarget.trans:=[9,34.0,0];
        MoveL pTarget,vSpeed,z0,tTool\WObj:=wWobj;
        pTarget.trans:=[7,31.0,0];
        MoveL pTarget,vSpeed,z0,tTool\WObj:=wWobj;
        pTarget.trans:=[5,27.0,0];
        MoveL pTarget,vSpeed,z0,tTool\WObj:=wWobj;
        pTarget.trans:=[4,22.0,0];
        MoveL pTarget,vSpeed,z0,tTool\WObj:=wWobj;
        pTarget.trans:=[4,18.0,0];
        MoveL pTarget,vSpeed,z0,tTool\WObj:=wWobj;
        pTarget.trans:=[5,13.0,0];
        MoveL pTarget,vSpeed,z0,tTool\WObj:=wWobj;
        pTarget.trans:=[7,9.0,0];
        MoveL pTarget,vSpeed,z0,tTool\WObj:=wWobj;
        pTarget.trans:=[9,6.0,0];
        MoveL pTarget,vSpeed,z0,tTool\WObj:=wWobj;
        pTarget.trans:=[11,4.0,0];
        MoveL pTarget,vSpeed,fine,tTool\WObj:=wWobj;
        Reset do_pen;
        MoveL RelTool(pTarget,0,0,-2),vSpeed,z0,tTool\WObj:=wWobj;
        wWobj.oframe.trans.x:=wWobj.oframe.trans.x+7;
    ENDPROC

    ! Character: )
    PROC char_rightparenthesis()
        VAR robtarget pTarget;
        pTarget:=refTarget;
        pTarget.trans:=[3,36.0,0];
        MoveL pTarget,vSpeed,fine,tTool\WObj:=wWobj;
        Set do_pen;
        pTarget.trans:=[5,34.0,0];
        MoveL pTarget,vSpeed,z0,tTool\WObj:=wWobj;
        pTarget.trans:=[7,31.0,0];
        MoveL pTarget,vSpeed,z0,tTool\WObj:=wWobj;
        pTarget.trans:=[9,27.0,0];
        MoveL pTarget,vSpeed,z0,tTool\WObj:=wWobj;
        pTarget.trans:=[10,22.0,0];
        MoveL pTarget,vSpeed,z0,tTool\WObj:=wWobj;
        pTarget.trans:=[10,18.0,0];
        MoveL pTarget,vSpeed,z0,tTool\WObj:=wWobj;
        pTarget.trans:=[9,13.0,0];
        MoveL pTarget,vSpeed,z0,tTool\WObj:=wWobj;
        pTarget.trans:=[7,9.0,0];
        MoveL pTarget,vSpeed,z0,tTool\WObj:=wWobj;
        pTarget.trans:=[5,6.0,0];
        MoveL pTarget,vSpeed,z0,tTool\WObj:=wWobj;
        pTarget.trans:=[3,4.0,0];
        MoveL pTarget,vSpeed,fine,tTool\WObj:=wWobj;
        Reset do_pen;
        MoveL RelTool(pTarget,0,0,-2),vSpeed,z0,tTool\WObj:=wWobj;
        wWobj.oframe.trans.x:=wWobj.oframe.trans.x+7;
    ENDPROC

    ! Character: +
    PROC char_plus()
        VAR robtarget pTarget;
        pTarget:=refTarget;
        pTarget.trans:=[13,29.0,0];
        MoveL pTarget,vSpeed,fine,tTool\WObj:=wWobj;
        Set do_pen;
        pTarget.trans:=[13,11.0,0];
        MoveL pTarget,vSpeed,fine,tTool\WObj:=wWobj;
        Reset do_pen;
        MoveL RelTool(pTarget,0,0,-2),vSpeed,z0,tTool\WObj:=wWobj;
        pTarget.trans:=[4,20.0,0];
        MoveL pTarget,vSpeed,fine,tTool\WObj:=wWobj;
        Set do_pen;
        pTarget.trans:=[22,20.0,0];
        MoveL pTarget,vSpeed,fine,tTool\WObj:=wWobj;
        Reset do_pen;
        MoveL RelTool(pTarget,0,0,-2),vSpeed,z0,tTool\WObj:=wWobj;
        wWobj.oframe.trans.x:=wWobj.oframe.trans.x+18;
    ENDPROC

    ! Character: =
    PROC char_equals()
        VAR robtarget pTarget;
        pTarget:=refTarget;
        pTarget.trans:=[4,23.0,0];
        MoveL pTarget,vSpeed,fine,tTool\WObj:=wWobj;
        Set do_pen;
        pTarget.trans:=[22,23.0,0];
        MoveL pTarget,vSpeed,fine,tTool\WObj:=wWobj;
        Reset do_pen;
        MoveL RelTool(pTarget,0,0,-2),vSpeed,z0,tTool\WObj:=wWobj;
        pTarget.trans:=[4,17.0,0];
        MoveL pTarget,vSpeed,fine,tTool\WObj:=wWobj;
        Set do_pen;
        pTarget.trans:=[22,17.0,0];
        MoveL pTarget,vSpeed,fine,tTool\WObj:=wWobj;
        Reset do_pen;
        MoveL RelTool(pTarget,0,0,-2),vSpeed,z0,tTool\WObj:=wWobj;
        wWobj.oframe.trans.x:=wWobj.oframe.trans.x+18;
    ENDPROC

    ! Character: [
    PROC char_leftbracket()
        VAR robtarget pTarget;
        pTarget:=refTarget;
        pTarget.trans:=[4,36.0,0];
        MoveL pTarget,vSpeed,fine,tTool\WObj:=wWobj;
        Set do_pen;
        pTarget.trans:=[4,4.0,0];
        MoveL pTarget,vSpeed,fine,tTool\WObj:=wWobj;
        Reset do_pen;
        MoveL RelTool(pTarget,0,0,-2),vSpeed,z0,tTool\WObj:=wWobj;
        pTarget.trans:=[5,36.0,0];
        MoveL pTarget,vSpeed,fine,tTool\WObj:=wWobj;
        Set do_pen;
        pTarget.trans:=[5,4.0,0];
        MoveL pTarget,vSpeed,fine,tTool\WObj:=wWobj;
        Reset do_pen;
        MoveL RelTool(pTarget,0,0,-2),vSpeed,z0,tTool\WObj:=wWobj;
        pTarget.trans:=[4,36.0,0];
        MoveL pTarget,vSpeed,fine,tTool\WObj:=wWobj;
        Set do_pen;
        pTarget.trans:=[11,36.0,0];
        MoveL pTarget,vSpeed,fine,tTool\WObj:=wWobj;
        Reset do_pen;
        MoveL RelTool(pTarget,0,0,-2),vSpeed,z0,tTool\WObj:=wWobj;
        pTarget.trans:=[4,4.0,0];
        MoveL pTarget,vSpeed,fine,tTool\WObj:=wWobj;
        Set do_pen;
        pTarget.trans:=[11,4.0,0];
        MoveL pTarget,vSpeed,fine,tTool\WObj:=wWobj;
        Reset do_pen;
        MoveL RelTool(pTarget,0,0,-2),vSpeed,z0,tTool\WObj:=wWobj;
        wWobj.oframe.trans.x:=wWobj.oframe.trans.x+7;
    ENDPROC

    ! Character: ]
    PROC char_rightbracket()
        VAR robtarget pTarget;
        pTarget:=refTarget;
        pTarget.trans:=[9,36.0,0];
        MoveL pTarget,vSpeed,fine,tTool\WObj:=wWobj;
        Set do_pen;
        pTarget.trans:=[9,4.0,0];
        MoveL pTarget,vSpeed,fine,tTool\WObj:=wWobj;
        Reset do_pen;
        MoveL RelTool(pTarget,0,0,-2),vSpeed,z0,tTool\WObj:=wWobj;
        pTarget.trans:=[10,36.0,0];
        MoveL pTarget,vSpeed,fine,tTool\WObj:=wWobj;
        Set do_pen;
        pTarget.trans:=[10,4.0,0];
        MoveL pTarget,vSpeed,fine,tTool\WObj:=wWobj;
        Reset do_pen;
        MoveL RelTool(pTarget,0,0,-2),vSpeed,z0,tTool\WObj:=wWobj;
        pTarget.trans:=[3,36.0,0];
        MoveL pTarget,vSpeed,fine,tTool\WObj:=wWobj;
        Set do_pen;
        pTarget.trans:=[10,36.0,0];
        MoveL pTarget,vSpeed,fine,tTool\WObj:=wWobj;
        Reset do_pen;
        MoveL RelTool(pTarget,0,0,-2),vSpeed,z0,tTool\WObj:=wWobj;
        pTarget.trans:=[3,4.0,0];
        MoveL pTarget,vSpeed,fine,tTool\WObj:=wWobj;
        Set do_pen;
        pTarget.trans:=[10,4.0,0];
        MoveL pTarget,vSpeed,fine,tTool\WObj:=wWobj;
        Reset do_pen;
        MoveL RelTool(pTarget,0,0,-2),vSpeed,z0,tTool\WObj:=wWobj;
        wWobj.oframe.trans.x:=wWobj.oframe.trans.x+7;
    ENDPROC

    ! Character: {
    PROC char_leftbrace()
        VAR robtarget pTarget;
        pTarget:=refTarget;
        pTarget.trans:=[9,36.0,0];
        MoveL pTarget,vSpeed,fine,tTool\WObj:=wWobj;
        Set do_pen;
        pTarget.trans:=[7,35.0,0];
        MoveL pTarget,vSpeed,z0,tTool\WObj:=wWobj;
        pTarget.trans:=[6,34.0,0];
        MoveL pTarget,vSpeed,z0,tTool\WObj:=wWobj;
        pTarget.trans:=[5,32.0,0];
        MoveL pTarget,vSpeed,z0,tTool\WObj:=wWobj;
        pTarget.trans:=[5,30.0,0];
        MoveL pTarget,vSpeed,z0,tTool\WObj:=wWobj;
        pTarget.trans:=[6,28.0,0];
        MoveL pTarget,vSpeed,z0,tTool\WObj:=wWobj;
        pTarget.trans:=[7,27.0,0];
        MoveL pTarget,vSpeed,z0,tTool\WObj:=wWobj;
        pTarget.trans:=[8,25.0,0];
        MoveL pTarget,vSpeed,z0,tTool\WObj:=wWobj;
        pTarget.trans:=[8,23.0,0];
        MoveL pTarget,vSpeed,z0,tTool\WObj:=wWobj;
        pTarget.trans:=[6,21.0,0];
        MoveL pTarget,vSpeed,fine,tTool\WObj:=wWobj;
        Reset do_pen;
        MoveL RelTool(pTarget,0,0,-2),vSpeed,z0,tTool\WObj:=wWobj;
        pTarget.trans:=[7,35.0,0];
        MoveL pTarget,vSpeed,fine,tTool\WObj:=wWobj;
        Set do_pen;
        pTarget.trans:=[6,33.0,0];
        MoveL pTarget,vSpeed,z0,tTool\WObj:=wWobj;
        pTarget.trans:=[6,31.0,0];
        MoveL pTarget,vSpeed,z0,tTool\WObj:=wWobj;
        pTarget.trans:=[7,29.0,0];
        MoveL pTarget,vSpeed,z0,tTool\WObj:=wWobj;
        pTarget.trans:=[8,28.0,0];
        MoveL pTarget,vSpeed,z0,tTool\WObj:=wWobj;
        pTarget.trans:=[9,26.0,0];
        MoveL pTarget,vSpeed,z0,tTool\WObj:=wWobj;
        pTarget.trans:=[9,24.0,0];
        MoveL pTarget,vSpeed,z0,tTool\WObj:=wWobj;
        pTarget.trans:=[8,22.0,0];
        MoveL pTarget,vSpeed,z0,tTool\WObj:=wWobj;
        pTarget.trans:=[4,20.0,0];
        MoveL pTarget,vSpeed,z0,tTool\WObj:=wWobj;
        pTarget.trans:=[8,18.0,0];
        MoveL pTarget,vSpeed,z0,tTool\WObj:=wWobj;
        pTarget.trans:=[9,16.0,0];
        MoveL pTarget,vSpeed,z0,tTool\WObj:=wWobj;
        pTarget.trans:=[9,14.0,0];
        MoveL pTarget,vSpeed,z0,tTool\WObj:=wWobj;
        pTarget.trans:=[8,12.0,0];
        MoveL pTarget,vSpeed,z0,tTool\WObj:=wWobj;
        pTarget.trans:=[7,11.0,0];
        MoveL pTarget,vSpeed,z0,tTool\WObj:=wWobj;
        pTarget.trans:=[6,9.0,0];
        MoveL pTarget,vSpeed,z0,tTool\WObj:=wWobj;
        pTarget.trans:=[6,7.0,0];
        MoveL pTarget,vSpeed,z0,tTool\WObj:=wWobj;
        pTarget.trans:=[7,5.0,0];
        MoveL pTarget,vSpeed,fine,tTool\WObj:=wWobj;
        Reset do_pen;
        MoveL RelTool(pTarget,0,0,-2),vSpeed,z0,tTool\WObj:=wWobj;
        pTarget.trans:=[6,19.0,0];
        MoveL pTarget,vSpeed,fine,tTool\WObj:=wWobj;
        Set do_pen;
        pTarget.trans:=[8,17.0,0];
        MoveL pTarget,vSpeed,z0,tTool\WObj:=wWobj;
        pTarget.trans:=[8,15.0,0];
        MoveL pTarget,vSpeed,z0,tTool\WObj:=wWobj;
        pTarget.trans:=[7,13.0,0];
        MoveL pTarget,vSpeed,z0,tTool\WObj:=wWobj;
        pTarget.trans:=[6,12.0,0];
        MoveL pTarget,vSpeed,z0,tTool\WObj:=wWobj;
        pTarget.trans:=[5,10.0,0];
        MoveL pTarget,vSpeed,z0,tTool\WObj:=wWobj;
        pTarget.trans:=[5,8.0,0];
        MoveL pTarget,vSpeed,z0,tTool\WObj:=wWobj;
        pTarget.trans:=[6,6.0,0];
        MoveL pTarget,vSpeed,z0,tTool\WObj:=wWobj;
        pTarget.trans:=[7,5.0,0];
        MoveL pTarget,vSpeed,z0,tTool\WObj:=wWobj;
        pTarget.trans:=[9,4.0,0];
        MoveL pTarget,vSpeed,fine,tTool\WObj:=wWobj;
        Reset do_pen;
        MoveL RelTool(pTarget,0,0,-2),vSpeed,z0,tTool\WObj:=wWobj;
        wWobj.oframe.trans.x:=wWobj.oframe.trans.x+5;
    ENDPROC

    ! Character: }
    PROC char_rightbrace()
        VAR robtarget pTarget;
        pTarget:=refTarget;
        pTarget.trans:=[5,36.0,0];
        MoveL pTarget,vSpeed,fine,tTool\WObj:=wWobj;
        Set do_pen;
        pTarget.trans:=[7,35.0,0];
        MoveL pTarget,vSpeed,z0,tTool\WObj:=wWobj;
        pTarget.trans:=[8,34.0,0];
        MoveL pTarget,vSpeed,z0,tTool\WObj:=wWobj;
        pTarget.trans:=[9,32.0,0];
        MoveL pTarget,vSpeed,z0,tTool\WObj:=wWobj;
        pTarget.trans:=[9,30.0,0];
        MoveL pTarget,vSpeed,z0,tTool\WObj:=wWobj;
        pTarget.trans:=[8,28.0,0];
        MoveL pTarget,vSpeed,z0,tTool\WObj:=wWobj;
        pTarget.trans:=[7,27.0,0];
        MoveL pTarget,vSpeed,z0,tTool\WObj:=wWobj;
        pTarget.trans:=[6,25.0,0];
        MoveL pTarget,vSpeed,z0,tTool\WObj:=wWobj;
        pTarget.trans:=[6,23.0,0];
        MoveL pTarget,vSpeed,z0,tTool\WObj:=wWobj;
        pTarget.trans:=[8,21.0,0];
        MoveL pTarget,vSpeed,fine,tTool\WObj:=wWobj;
        Reset do_pen;
        MoveL RelTool(pTarget,0,0,-2),vSpeed,z0,tTool\WObj:=wWobj;
        pTarget.trans:=[7,35.0,0];
        MoveL pTarget,vSpeed,fine,tTool\WObj:=wWobj;
        Set do_pen;
        pTarget.trans:=[8,33.0,0];
        MoveL pTarget,vSpeed,z0,tTool\WObj:=wWobj;
        pTarget.trans:=[8,31.0,0];
        MoveL pTarget,vSpeed,z0,tTool\WObj:=wWobj;
        pTarget.trans:=[7,29.0,0];
        MoveL pTarget,vSpeed,z0,tTool\WObj:=wWobj;
        pTarget.trans:=[6,28.0,0];
        MoveL pTarget,vSpeed,z0,tTool\WObj:=wWobj;
        pTarget.trans:=[5,26.0,0];
        MoveL pTarget,vSpeed,z0,tTool\WObj:=wWobj;
        pTarget.trans:=[5,24.0,0];
        MoveL pTarget,vSpeed,z0,tTool\WObj:=wWobj;
        pTarget.trans:=[6,22.0,0];
        MoveL pTarget,vSpeed,z0,tTool\WObj:=wWobj;
        pTarget.trans:=[10,20.0,0];
        MoveL pTarget,vSpeed,z0,tTool\WObj:=wWobj;
        pTarget.trans:=[6,18.0,0];
        MoveL pTarget,vSpeed,z0,tTool\WObj:=wWobj;
        pTarget.trans:=[5,16.0,0];
        MoveL pTarget,vSpeed,z0,tTool\WObj:=wWobj;
        pTarget.trans:=[5,14.0,0];
        MoveL pTarget,vSpeed,z0,tTool\WObj:=wWobj;
        pTarget.trans:=[6,12.0,0];
        MoveL pTarget,vSpeed,z0,tTool\WObj:=wWobj;
        pTarget.trans:=[7,11.0,0];
        MoveL pTarget,vSpeed,z0,tTool\WObj:=wWobj;
        pTarget.trans:=[8,9.0,0];
        MoveL pTarget,vSpeed,z0,tTool\WObj:=wWobj;
        pTarget.trans:=[8,7.0,0];
        MoveL pTarget,vSpeed,z0,tTool\WObj:=wWobj;
        pTarget.trans:=[7,5.0,0];
        MoveL pTarget,vSpeed,fine,tTool\WObj:=wWobj;
        Reset do_pen;
        MoveL RelTool(pTarget,0,0,-2),vSpeed,z0,tTool\WObj:=wWobj;
        pTarget.trans:=[8,19.0,0];
        MoveL pTarget,vSpeed,fine,tTool\WObj:=wWobj;
        Set do_pen;
        pTarget.trans:=[6,17.0,0];
        MoveL pTarget,vSpeed,z0,tTool\WObj:=wWobj;
        pTarget.trans:=[6,15.0,0];
        MoveL pTarget,vSpeed,z0,tTool\WObj:=wWobj;
        pTarget.trans:=[7,13.0,0];
        MoveL pTarget,vSpeed,z0,tTool\WObj:=wWobj;
        pTarget.trans:=[8,12.0,0];
        MoveL pTarget,vSpeed,z0,tTool\WObj:=wWobj;
        pTarget.trans:=[9,10.0,0];
        MoveL pTarget,vSpeed,z0,tTool\WObj:=wWobj;
        pTarget.trans:=[9,8.0,0];
        MoveL pTarget,vSpeed,z0,tTool\WObj:=wWobj;
        pTarget.trans:=[8,6.0,0];
        MoveL pTarget,vSpeed,z0,tTool\WObj:=wWobj;
        pTarget.trans:=[7,5.0,0];
        MoveL pTarget,vSpeed,z0,tTool\WObj:=wWobj;
        pTarget.trans:=[5,4.0,0];
        MoveL pTarget,vSpeed,fine,tTool\WObj:=wWobj;
        Reset do_pen;
        MoveL RelTool(pTarget,0,0,-2),vSpeed,z0,tTool\WObj:=wWobj;
        wWobj.oframe.trans.x:=wWobj.oframe.trans.x+5;
    ENDPROC

    ! Character: |
    PROC char_pipe()
        VAR robtarget pTarget;
        pTarget:=refTarget;
        pTarget.trans:=[4,36.0,0];
        MoveL pTarget,vSpeed,fine,tTool\WObj:=wWobj;
        Set do_pen;
        pTarget.trans:=[4,4.0,0];
        MoveL pTarget,vSpeed,fine,tTool\WObj:=wWobj;
        Reset do_pen;
        MoveL RelTool(pTarget,0,0,-2),vSpeed,z0,tTool\WObj:=wWobj;
        wWobj.oframe.trans.x:=wWobj.oframe.trans.x+1.0;
    ENDPROC

    ! Character: <
    PROC char_lessthan()
        VAR robtarget pTarget;
        pTarget:=refTarget;
        pTarget.trans:=[20,29.0,0];
        MoveL pTarget,vSpeed,fine,tTool\WObj:=wWobj;
        Set do_pen;
        pTarget.trans:=[4,20.0,0];
        MoveL pTarget,vSpeed,z0,tTool\WObj:=wWobj;
        pTarget.trans:=[20,11.0,0];
        MoveL pTarget,vSpeed,fine,tTool\WObj:=wWobj;
        Reset do_pen;
        MoveL RelTool(pTarget,0,0,-2),vSpeed,z0,tTool\WObj:=wWobj;
        wWobj.oframe.trans.x:=wWobj.oframe.trans.x+16;
    ENDPROC

    ! Character: >
    PROC char_greaterthan()
        VAR robtarget pTarget;
        pTarget:=refTarget;
        pTarget.trans:=[4,29.0,0];
        MoveL pTarget,vSpeed,fine,tTool\WObj:=wWobj;
        Set do_pen;
        pTarget.trans:=[20,20.0,0];
        MoveL pTarget,vSpeed,z0,tTool\WObj:=wWobj;
        pTarget.trans:=[4,11.0,0];
        MoveL pTarget,vSpeed,fine,tTool\WObj:=wWobj;
        Reset do_pen;
        MoveL RelTool(pTarget,0,0,-2),vSpeed,z0,tTool\WObj:=wWobj;
        wWobj.oframe.trans.x:=wWobj.oframe.trans.x+16;
    ENDPROC

    ! Character: ?
    PROC char_question()
        VAR robtarget pTarget;
        pTarget:=refTarget;
        pTarget.trans:=[3,27.0,0];
        MoveL pTarget,vSpeed,fine,tTool\WObj:=wWobj;
        Set do_pen;
        pTarget.trans:=[3,28.0,0];
        MoveL pTarget,vSpeed,z0,tTool\WObj:=wWobj;
        pTarget.trans:=[4,30.0,0];
        MoveL pTarget,vSpeed,z0,tTool\WObj:=wWobj;
        pTarget.trans:=[5,31.0,0];
        MoveL pTarget,vSpeed,z0,tTool\WObj:=wWobj;
        pTarget.trans:=[7,32.0,0];
        MoveL pTarget,vSpeed,z0,tTool\WObj:=wWobj;
        pTarget.trans:=[11,32.0,0];
        MoveL pTarget,vSpeed,z0,tTool\WObj:=wWobj;
        pTarget.trans:=[13,31.0,0];
        MoveL pTarget,vSpeed,z0,tTool\WObj:=wWobj;
        pTarget.trans:=[14,30.0,0];
        MoveL pTarget,vSpeed,z0,tTool\WObj:=wWobj;
        pTarget.trans:=[15,28.0,0];
        MoveL pTarget,vSpeed,z0,tTool\WObj:=wWobj;
        pTarget.trans:=[15,26.0,0];
        MoveL pTarget,vSpeed,z0,tTool\WObj:=wWobj;
        pTarget.trans:=[14,24.0,0];
        MoveL pTarget,vSpeed,z0,tTool\WObj:=wWobj;
        pTarget.trans:=[13,23.0,0];
        MoveL pTarget,vSpeed,z0,tTool\WObj:=wWobj;
        pTarget.trans:=[9,21.0,0];
        MoveL pTarget,vSpeed,z0,tTool\WObj:=wWobj;
        pTarget.trans:=[9,18.0,0];
        MoveL pTarget,vSpeed,fine,tTool\WObj:=wWobj;
        Reset do_pen;
        MoveL RelTool(pTarget,0,0,-2),vSpeed,z0,tTool\WObj:=wWobj;
        pTarget.trans:=[9,13.0,0];
        MoveL pTarget,vSpeed,fine,tTool\WObj:=wWobj;
        Set do_pen;
        pTarget.trans:=[8,12.0,0];
        MoveL pTarget,vSpeed,z0,tTool\WObj:=wWobj;
        pTarget.trans:=[9,11.0,0];
        MoveL pTarget,vSpeed,z0,tTool\WObj:=wWobj;
        pTarget.trans:=[10,12.0,0];
        MoveL pTarget,vSpeed,z0,tTool\WObj:=wWobj;
        pTarget.trans:=[9,13.0,0];
        MoveL pTarget,vSpeed,fine,tTool\WObj:=wWobj;
        Reset do_pen;
        MoveL RelTool(pTarget,0,0,-2),vSpeed,z0,tTool\WObj:=wWobj;
        wWobj.oframe.trans.x:=wWobj.oframe.trans.x+12;
    ENDPROC

    ! Character: _
    PROC char_underscore()
        VAR robtarget pTarget;
        pTarget:=refTarget;
        pTarget.trans:=[0,4.0,0];
        MoveL pTarget,vSpeed,fine,tTool\WObj:=wWobj;
        Set do_pen;
        pTarget.trans:=[20,4.0,0];
        MoveL pTarget,vSpeed,fine,tTool\WObj:=wWobj;
        Reset do_pen;
        MoveL RelTool(pTarget,0,0,-2),vSpeed,z0,tTool\WObj:=wWobj;
        wWobj.oframe.trans.x:=wWobj.oframe.trans.x+20;
    ENDPROC

    ! Character: -
    PROC char_minus()
        VAR robtarget pTarget;
        pTarget:=refTarget;
        pTarget.trans:=[4,20.0,0];
        MoveL pTarget,vSpeed,fine,tTool\WObj:=wWobj;
        Set do_pen;
        pTarget.trans:=[22,20.0,0];
        MoveL pTarget,vSpeed,fine,tTool\WObj:=wWobj;
        Reset do_pen;
        MoveL RelTool(pTarget,0,0,-2),vSpeed,z0,tTool\WObj:=wWobj;
        wWobj.oframe.trans.x:=wWobj.oframe.trans.x+18;
    ENDPROC

    ! Character: ~
    PROC char_tilde()
        VAR robtarget pTarget;
        pTarget:=refTarget;
        pTarget.trans:=[3,17.0,0];
        MoveL pTarget,vSpeed,fine,tTool\WObj:=wWobj;
        Set do_pen;
        pTarget.trans:=[3,19.0,0];
        MoveL pTarget,vSpeed,z0,tTool\WObj:=wWobj;
        pTarget.trans:=[4,22.0,0];
        MoveL pTarget,vSpeed,z0,tTool\WObj:=wWobj;
        pTarget.trans:=[6,23.0,0];
        MoveL pTarget,vSpeed,z0,tTool\WObj:=wWobj;
        pTarget.trans:=[8,23.0,0];
        MoveL pTarget,vSpeed,z0,tTool\WObj:=wWobj;
        pTarget.trans:=[10,22.0,0];
        MoveL pTarget,vSpeed,z0,tTool\WObj:=wWobj;
        pTarget.trans:=[14,19.0,0];
        MoveL pTarget,vSpeed,z0,tTool\WObj:=wWobj;
        pTarget.trans:=[16,18.0,0];
        MoveL pTarget,vSpeed,z0,tTool\WObj:=wWobj;
        pTarget.trans:=[18,18.0,0];
        MoveL pTarget,vSpeed,z0,tTool\WObj:=wWobj;
        pTarget.trans:=[20,19.0,0];
        MoveL pTarget,vSpeed,z0,tTool\WObj:=wWobj;
        pTarget.trans:=[21,21.0,0];
        MoveL pTarget,vSpeed,fine,tTool\WObj:=wWobj;
        Reset do_pen;
        MoveL RelTool(pTarget,0,0,-2),vSpeed,z0,tTool\WObj:=wWobj;
        pTarget.trans:=[3,19.0,0];
        MoveL pTarget,vSpeed,fine,tTool\WObj:=wWobj;
        Set do_pen;
        pTarget.trans:=[4,21.0,0];
        MoveL pTarget,vSpeed,z0,tTool\WObj:=wWobj;
        pTarget.trans:=[6,22.0,0];
        MoveL pTarget,vSpeed,z0,tTool\WObj:=wWobj;
        pTarget.trans:=[8,22.0,0];
        MoveL pTarget,vSpeed,z0,tTool\WObj:=wWobj;
        pTarget.trans:=[10,21.0,0];
        MoveL pTarget,vSpeed,z0,tTool\WObj:=wWobj;
        pTarget.trans:=[14,18.0,0];
        MoveL pTarget,vSpeed,z0,tTool\WObj:=wWobj;
        pTarget.trans:=[16,17.0,0];
        MoveL pTarget,vSpeed,z0,tTool\WObj:=wWobj;
        pTarget.trans:=[18,17.0,0];
        MoveL pTarget,vSpeed,z0,tTool\WObj:=wWobj;
        pTarget.trans:=[20,18.0,0];
        MoveL pTarget,vSpeed,z0,tTool\WObj:=wWobj;
        pTarget.trans:=[21,21.0,0];
        MoveL pTarget,vSpeed,z0,tTool\WObj:=wWobj;
        pTarget.trans:=[21,23.0,0];
        MoveL pTarget,vSpeed,fine,tTool\WObj:=wWobj;
        Reset do_pen;
        MoveL RelTool(pTarget,0,0,-2),vSpeed,z0,tTool\WObj:=wWobj;
        wWobj.oframe.trans.x:=wWobj.oframe.trans.x+18;
    ENDPROC

    ! Character: .
    PROC char_period()
        VAR robtarget pTarget;
        pTarget:=refTarget;
        pTarget.trans:=[4,16.0,0];
        MoveL pTarget,vSpeed,fine,tTool\WObj:=wWobj;
        Set do_pen;
        pTarget.trans:=[3,15.0,0];
        MoveL pTarget,vSpeed,z0,tTool\WObj:=wWobj;
        pTarget.trans:=[4,14.0,0];
        MoveL pTarget,vSpeed,z0,tTool\WObj:=wWobj;
        pTarget.trans:=[5,15.0,0];
        MoveL pTarget,vSpeed,z0,tTool\WObj:=wWobj;
        pTarget.trans:=[4,16.0,0];
        MoveL pTarget,vSpeed,fine,tTool\WObj:=wWobj;
        Reset do_pen;
        MoveL RelTool(pTarget,0,0,-2),vSpeed,z0,tTool\WObj:=wWobj;
        wWobj.oframe.trans.x:=wWobj.oframe.trans.x+2;
    ENDPROC

    ! Character: ,
    PROC char_comma()
        VAR robtarget pTarget;
        pTarget:=refTarget;
        pTarget.trans:=[5,15.0,0];
        MoveL pTarget,vSpeed,fine,tTool\WObj:=wWobj;
        Set do_pen;
        pTarget.trans:=[4,14.0,0];
        MoveL pTarget,vSpeed,z0,tTool\WObj:=wWobj;
        pTarget.trans:=[3,15.0,0];
        MoveL pTarget,vSpeed,z0,tTool\WObj:=wWobj;
        pTarget.trans:=[4,16.0,0];
        MoveL pTarget,vSpeed,z0,tTool\WObj:=wWobj;
        pTarget.trans:=[5,15.0,0];
        MoveL pTarget,vSpeed,z0,tTool\WObj:=wWobj;
        pTarget.trans:=[5,13.0,0];
        MoveL pTarget,vSpeed,z0,tTool\WObj:=wWobj;
        pTarget.trans:=[3,11.0,0];
        MoveL pTarget,vSpeed,fine,tTool\WObj:=wWobj;
        Reset do_pen;
        MoveL RelTool(pTarget,0,0,-2),vSpeed,z0,tTool\WObj:=wWobj;
        wWobj.oframe.trans.x:=wWobj.oframe.trans.x+2;
    ENDPROC

    ! Character: ;
    PROC char_semicolon()
        VAR robtarget pTarget;
        pTarget:=refTarget;
        pTarget.trans:=[4,23.0,0];
        MoveL pTarget,vSpeed,fine,tTool\WObj:=wWobj;
        Set do_pen;
        pTarget.trans:=[3,22.0,0];
        MoveL pTarget,vSpeed,z0,tTool\WObj:=wWobj;
        pTarget.trans:=[4,21.0,0];
        MoveL pTarget,vSpeed,z0,tTool\WObj:=wWobj;
        pTarget.trans:=[5,22.0,0];
        MoveL pTarget,vSpeed,z0,tTool\WObj:=wWobj;
        pTarget.trans:=[4,23.0,0];
        MoveL pTarget,vSpeed,fine,tTool\WObj:=wWobj;
        Reset do_pen;
        MoveL RelTool(pTarget,0,0,-2),vSpeed,z0,tTool\WObj:=wWobj;
        pTarget.trans:=[5,15.0,0];
        MoveL pTarget,vSpeed,fine,tTool\WObj:=wWobj;
        Set do_pen;
        pTarget.trans:=[4,14.0,0];
        MoveL pTarget,vSpeed,z0,tTool\WObj:=wWobj;
        pTarget.trans:=[3,15.0,0];
        MoveL pTarget,vSpeed,z0,tTool\WObj:=wWobj;
        pTarget.trans:=[4,16.0,0];
        MoveL pTarget,vSpeed,z0,tTool\WObj:=wWobj;
        pTarget.trans:=[5,15.0,0];
        MoveL pTarget,vSpeed,z0,tTool\WObj:=wWobj;
        pTarget.trans:=[5,13.0,0];
        MoveL pTarget,vSpeed,z0,tTool\WObj:=wWobj;
        pTarget.trans:=[3,11.0,0];
        MoveL pTarget,vSpeed,fine,tTool\WObj:=wWobj;
        Reset do_pen;
        MoveL RelTool(pTarget,0,0,-2),vSpeed,z0,tTool\WObj:=wWobj;
        wWobj.oframe.trans.x:=wWobj.oframe.trans.x+2;
    ENDPROC

    ! Character: :
    PROC char_colon()
        VAR robtarget pTarget;
        pTarget:=refTarget;
        pTarget.trans:=[4,23.0,0];
        MoveL pTarget,vSpeed,fine,tTool\WObj:=wWobj;
        Set do_pen;
        pTarget.trans:=[3,22.0,0];
        MoveL pTarget,vSpeed,z0,tTool\WObj:=wWobj;
        pTarget.trans:=[4,21.0,0];
        MoveL pTarget,vSpeed,z0,tTool\WObj:=wWobj;
        pTarget.trans:=[5,22.0,0];
        MoveL pTarget,vSpeed,z0,tTool\WObj:=wWobj;
        pTarget.trans:=[4,23.0,0];
        MoveL pTarget,vSpeed,fine,tTool\WObj:=wWobj;
        Reset do_pen;
        MoveL RelTool(pTarget,0,0,-2),vSpeed,z0,tTool\WObj:=wWobj;
        pTarget.trans:=[4,16.0,0];
        MoveL pTarget,vSpeed,fine,tTool\WObj:=wWobj;
        Set do_pen;
        pTarget.trans:=[3,15.0,0];
        MoveL pTarget,vSpeed,z0,tTool\WObj:=wWobj;
        pTarget.trans:=[4,14.0,0];
        MoveL pTarget,vSpeed,z0,tTool\WObj:=wWobj;
        pTarget.trans:=[5,15.0,0];
        MoveL pTarget,vSpeed,z0,tTool\WObj:=wWobj;
        pTarget.trans:=[4,16.0,0];
        MoveL pTarget,vSpeed,fine,tTool\WObj:=wWobj;
        Reset do_pen;
        MoveL RelTool(pTarget,0,0,-2),vSpeed,z0,tTool\WObj:=wWobj;
        wWobj.oframe.trans.x:=wWobj.oframe.trans.x+2;
    ENDPROC
ENDMODULE

--- Controller Data/IRB1200_5_90/RAPID/TASK1/PROGMOD/Module1.modx ---
MODULE Module1
    PERS tooldata tTool:=[TRUE,[[110,0,140],[0.707106781,0,0.707106781,0]],[1,[10.7435139,0,140],[1,0,0,0],0,0,0]];
    PERS wobjdata wWobj:=[FALSE,TRUE,"",[[526.92,-115.652,257.517],[0.695575,0.127182,0.127182,0.695575]],[[235,110,1],[1,0,0,0]]];
    VAR speeddata vSpeed:=[150,3000,100,3000];
    PERS tooldata Pen_TCP:=[TRUE,[[110,0,140],[0.707106781,0,0.707106781,0]],[1,[10.7435139,0,140],[1,0,0,0],0,0,0]];
    CONST robtarget refTarget:=[[-61.41097207,14.187566617,-0.240748359],[0.098541688,-0.538960856,-0.836538911,-0.00365808],[-1,-1,0,1],[9E+09,9E+09,9E+09,9E+09,9E+09,9E+09]];

    PROC main()
        VAR robtarget pNow;
        reset do_pen;
        wWobj.oframe.trans.z:=1;
        wWobj.oframe.trans.y:=150;
        wWobj.oframe.trans.x:=wobj0.oframe.trans.x+20;
        WriteCursive "Salut Aurelien!";
        pNow:=CRobT();
        MoveL RelTool(pNow,0,0,-40),vmax,fine,tTool\wobj:=wWobj;
        reset do_pen;
        wWobj.oframe.trans.y:=110;
        wWobj.oframe.trans.x:=wobj0.oframe.trans.x+20;
        WriteCursive "Te souviens-tu ?";
        pNow:=CRobT();
        MoveL RelTool(pNow,0,0,-40),vmax,fine,tTool\wobj:=wWobj;
    ENDPROC

